// TIA Portal V20 export
FUNCTION_BLOCK "Sequence_2_SepaGripper"   // FB228, LAD
AUTHOR : ERsystem_FA2_DH. Kim
// stored: IsIECCheckEnabled true, MemoryReserve 100, Namespace Unit1.Em7, SetENOAutomatically false
   VAR_INPUT
      unitStatus { ExternalAccessible := 'False'; ExternalVisible := 'False'; ExternalWritable := 'False'} : "LAF_typeUnitStatus";   // Current unit status o be used in this EM
   END_VAR
   VAR
      statSelectedJobNumber { ExternalWritable := 'False'} : DInt;   // Evaluated Job Number
      instSequenceLADStatus { ExternalWritable := 'False'} : "LAF_StatusLadSequence";
      instSequenceLADControl { ExternalWritable := 'False'} : "LAF_ControlLadSequence";
      statTonTime { ExternalAccessible := 'False'; ExternalVisible := 'False'; ExternalWritable := 'False'} : Array[0..999] of TON_TIME;
   END_VAR
   VAR CONSTANT
      STEP_IDLE : DInt := 1;
      STEP_IMMEDIATE_STOP : DInt := 9001;   // Step executed when an immediate stop command is triggered for the sequence (i.e. when unit is in state aborting)
      JOB_1_STEP_01 : DInt := 101;
      JOB_1_STEP_10 : DInt := 110;
      JOB_1_STEP_20 : DInt := 120;
      JOB_1_STEP_30 : DInt := 130;
      JOB_1_STEP_40 : DInt := 140;
      JOB_1_STEP_41 : DInt := 141;
      JOB_1_STEP_50 : DInt := 150;
      JOB_1_STEP_80 : DInt := 180;
      JOB_1_STEP_90 : DInt := 190;
      JOB_2_STEP_01 : DInt := 201;
      JOB_2_STEP_10 : DInt := 210;
      JOB_2_STEP_20 : DInt := 220;
      JOB_2_STEP_30 : DInt := 230;
      JOB_2_STEP_31 : DInt := 231;
      JOB_2_STEP_40 : DInt := 240;
      JOB_2_STEP_50 : DInt := 250;
      JOB_2_STEP_51 : DInt := 251;
      JOB_2_STEP_80 : DInt := 280;
      JOB_2_STEP_90 : DInt := 290;
      JOB_3_STEP_01 : DInt := 301;
      JOB_3_STEP_10 : DInt := 310;
      JOB_3_STEP_11 : DInt := 311;
      JOB_3_STEP_20 : DInt := 320;
      JOB_3_STEP_30 : DInt := 330;
      JOB_3_STEP_31 : DInt := 331;
      JOB_3_STEP_90 : DInt := 390;
      JOB_4_STEP_01 : DInt := 401;
      JOB_4_STEP_10 : DInt := 410;
      JOB_4_STEP_20 : DInt := 420;
      JOB_4_STEP_21 : DInt := 421;
      JOB_4_STEP_30 : DInt := 430;
      JOB_4_STEP_90 : DInt := 490;
      JOB_5_STEP_01 : DInt := 501;
      JOB_5_STEP_10 : DInt := 510;
      JOB_5_STEP_20 : DInt := 520;
      JOB_5_STEP_30 : DInt := 530;
      JOB_5_STEP_31 : DInt := 531;
      JOB_5_STEP_40 : DInt := 540;
      JOB_5_STEP_50 : DInt := 550;
      JOB_5_STEP_80 : DInt := 580;
      JOB_5_STEP_81 : DInt := 581;
      JOB_5_STEP_90 : DInt := 590;
      JOB_6_STEP_01 : DInt := 601;
      JOB_6_STEP_10 : DInt := 610;
      JOB_6_STEP_11 : DInt := 611;
      JOB_6_STEP_20 : DInt := 620;
      JOB_6_STEP_90 : DInt := 690;
      JOB_7_STEP_01 : DInt := 701;
      JOB_7_STEP_10 : DInt := 710;
      JOB_7_STEP_20 : DInt := 720;
      JOB_7_STEP_30 : DInt := 730;
      JOB_7_STEP_40 : DInt := 740;
      JOB_7_STEP_50 : DInt := 750;
      JOB_7_STEP_90 : DInt := 790;
      JOB_8_STEP_01 : DInt := 801;
      JOB_8_STEP_10 : DInt := 810;
      JOB_8_STEP_11 : DInt := 811;
      JOB_8_STEP_20 : DInt := 820;
      JOB_8_STEP_21 : DInt := 821;
      JOB_8_STEP_30 : DInt := 830;
      JOB_8_STEP_31 : DInt := 831;
      JOB_8_STEP_90 : DInt := 890;
      JOB_9_STEP_01 : DInt := 901;
      JOB_9_STEP_10 : DInt := 910;
      JOB_9_STEP_20 : DInt := 920;
      JOB_9_STEP_30 : DInt := 930;
      JOB_9_STEP_40 : DInt := 940;
      JOB_9_STEP_50 : DInt := 950;
      JOB_9_STEP_90 : DInt := 990;
      JOB_11_STEP_01 : DInt := 1101;
      JOB_11_STEP_10 : DInt := 1110;
      JOB_11_STEP_20 : DInt := 1120;
      JOB_11_STEP_30 : DInt := 1130;
      JOB_11_STEP_40 : DInt := 1140;
      JOB_11_STEP_90 : DInt := 1190;
      JOB_12_STEP_01 : DInt := 1201;
      JOB_12_STEP_10 : DInt := 1210;
      JOB_12_STEP_11 : DInt := 1211;
      JOB_12_STEP_15 : DInt := 1215;
      JOB_12_STEP_16 : DInt := 1216;
      JOB_12_STEP_20 : DInt := 1220;
      JOB_12_STEP_30 : DInt := 1230;
      JOB_12_STEP_40 : DInt := 1240;
      JOB_12_STEP_90 : DInt := 1290;
      JOB_13_STEP_01 : DInt := 1301;
      JOB_13_STEP_10 : DInt := 1310;
      JOB_13_STEP_11 : DInt := 1311;
      JOB_13_STEP_90 : DInt := 1390;
      JOB_14_STEP_01 : DInt := 1401;
      JOB_14_STEP_10 : DInt := 1410;
      JOB_14_STEP_20 : DInt := 1420;
      JOB_14_STEP_90 : DInt := 1490;
      JOB_15_STEP_01 : DInt := 1501;
      JOB_15_STEP_10 : DInt := 1510;
      JOB_15_STEP_11 : DInt := 1511;
      JOB_15_STEP_20 : DInt := 1520;
      JOB_15_STEP_25 : DInt := 1525;
      JOB_15_STEP_30 : DInt := 1530;
      JOB_15_STEP_40 : DInt := 1540;
      JOB_15_STEP_50 : DInt := 1550;
      JOB_15_STEP_60 : DInt := 1560;
      JOB_15_STEP_70 : DInt := 1570;
      JOB_15_STEP_90 : DInt := 1590;
      JOB_16_STEP_01 : DInt := 1601;
      JOB_16_STEP_10 : DInt := 1610;
      JOB_16_STEP_20 : DInt := 1620;
      JOB_16_STEP_30 : DInt := 1630;
      JOB_16_STEP_40 : DInt := 1640;
      JOB_16_STEP_50 : DInt := 1650;
      JOB_16_STEP_90 : DInt := 1690;
      JOB_17_STEP_01 : DInt := 1701;
      JOB_17_STEP_10 : DInt := 1710;
      JOB_17_STEP_11 : DInt := 1711;
      JOB_17_STEP_20 : DInt := 1720;
      JOB_17_STEP_21 : DInt := 1721;
      JOB_17_STEP_30 : DInt := 1730;
      JOB_17_STEP_31 : DInt := 1731;
      JOB_17_STEP_90 : DInt := 1790;
      JOB_18_STEP_01 : DInt := 1801;
      JOB_18_STEP_10 : DInt := 1810;
      JOB_18_STEP_20 : DInt := 1820;
      JOB_18_STEP_30 : DInt := 1830;
      JOB_18_STEP_40 : DInt := 1840;
      JOB_18_STEP_50 : DInt := 1850;
      JOB_18_STEP_90 : DInt := 1890;
      FALSE : Bool := FALSE;
      TRUE : Bool := TRUE;
   END_VAR
   VAR_TEMP   // added for the SCL form of the ladder/FBD networks
      _w1 : Bool;
      _w2 : Bool;
   END_VAR
BEGIN

REGION Network 1: BLOCK INFO HEADER
   // (company) / (C) Copyright (year)
   // ---------------------------------------------------------------------------------
   // Title:                             (Title of this block)
   // Comment/Function: (that is implemented in the block)
   // Library/Family:           (that the source is dedicated to)
   // Author:                        (department / person in charge / contact)
   // Target System:          (test system with FW version)
   // Engineering:              TIA Portal (SW version)
   // Restrictions:               (OB types, etc.)
   // Requirements:           (hardware, technological package, etc.)
   // ---------------------------------------------------------------------------------
   // Change log table:
   // Version          | Date             | Signature      | Expert in charge  | Changes applied ------------------------|----------------------|-------------------------|--------------------------------|-----------------------
   // 001.000.000 | yyyy-mm-dd | 0x00000000 | (name of expert) | First released version
END_REGION

REGION Network 2: DESCRIPTION
   // This is a template block provided by the Automation Framework. It can be used to create an own project.
   // The Block Info Header is prepared to put in your own data.
   // Description of the block could be added here and the docu created by Code2Docu.
END_REGION

REGION Network 3: ********************* CONTROL *************************
END_REGION

REGION Network 4: Sequence Control
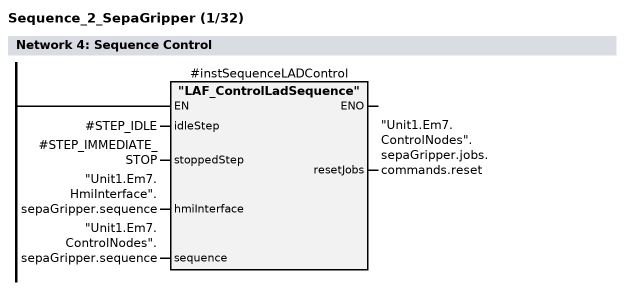
   RUNG wire#powerrail
      #instSequenceLADControl(idleStep := #STEP_IDLE, stoppedStep := #STEP_IMMEDIATE_STOP, hmiInterface := "Unit1.Em7.HmiInterface".sepaGripper.sequence, sequence := "Unit1.Em7.ControlNodes".sepaGripper.sequence, resetJobs => "Unit1.Em7.ControlNodes".sepaGripper.jobs.commands.reset)
   END_RUNG
   // the same network as SCL:
   #instSequenceLADControl(idleStep := #STEP_IDLE,   // "LAF_ControlLadSequence"
                           stoppedStep := #STEP_IMMEDIATE_STOP,
                           hmiInterface := "Unit1.Em7.HmiInterface".sepaGripper.sequence,
                           sequence := "Unit1.Em7.ControlNodes".sepaGripper.sequence,
                           resetJobs => "Unit1.Em7.ControlNodes".sepaGripper.jobs.commands.reset);
END_REGION

REGION Network 5: *************** JOB SELECT **************************
END_REGION

REGION Network 6: STEP IDLE
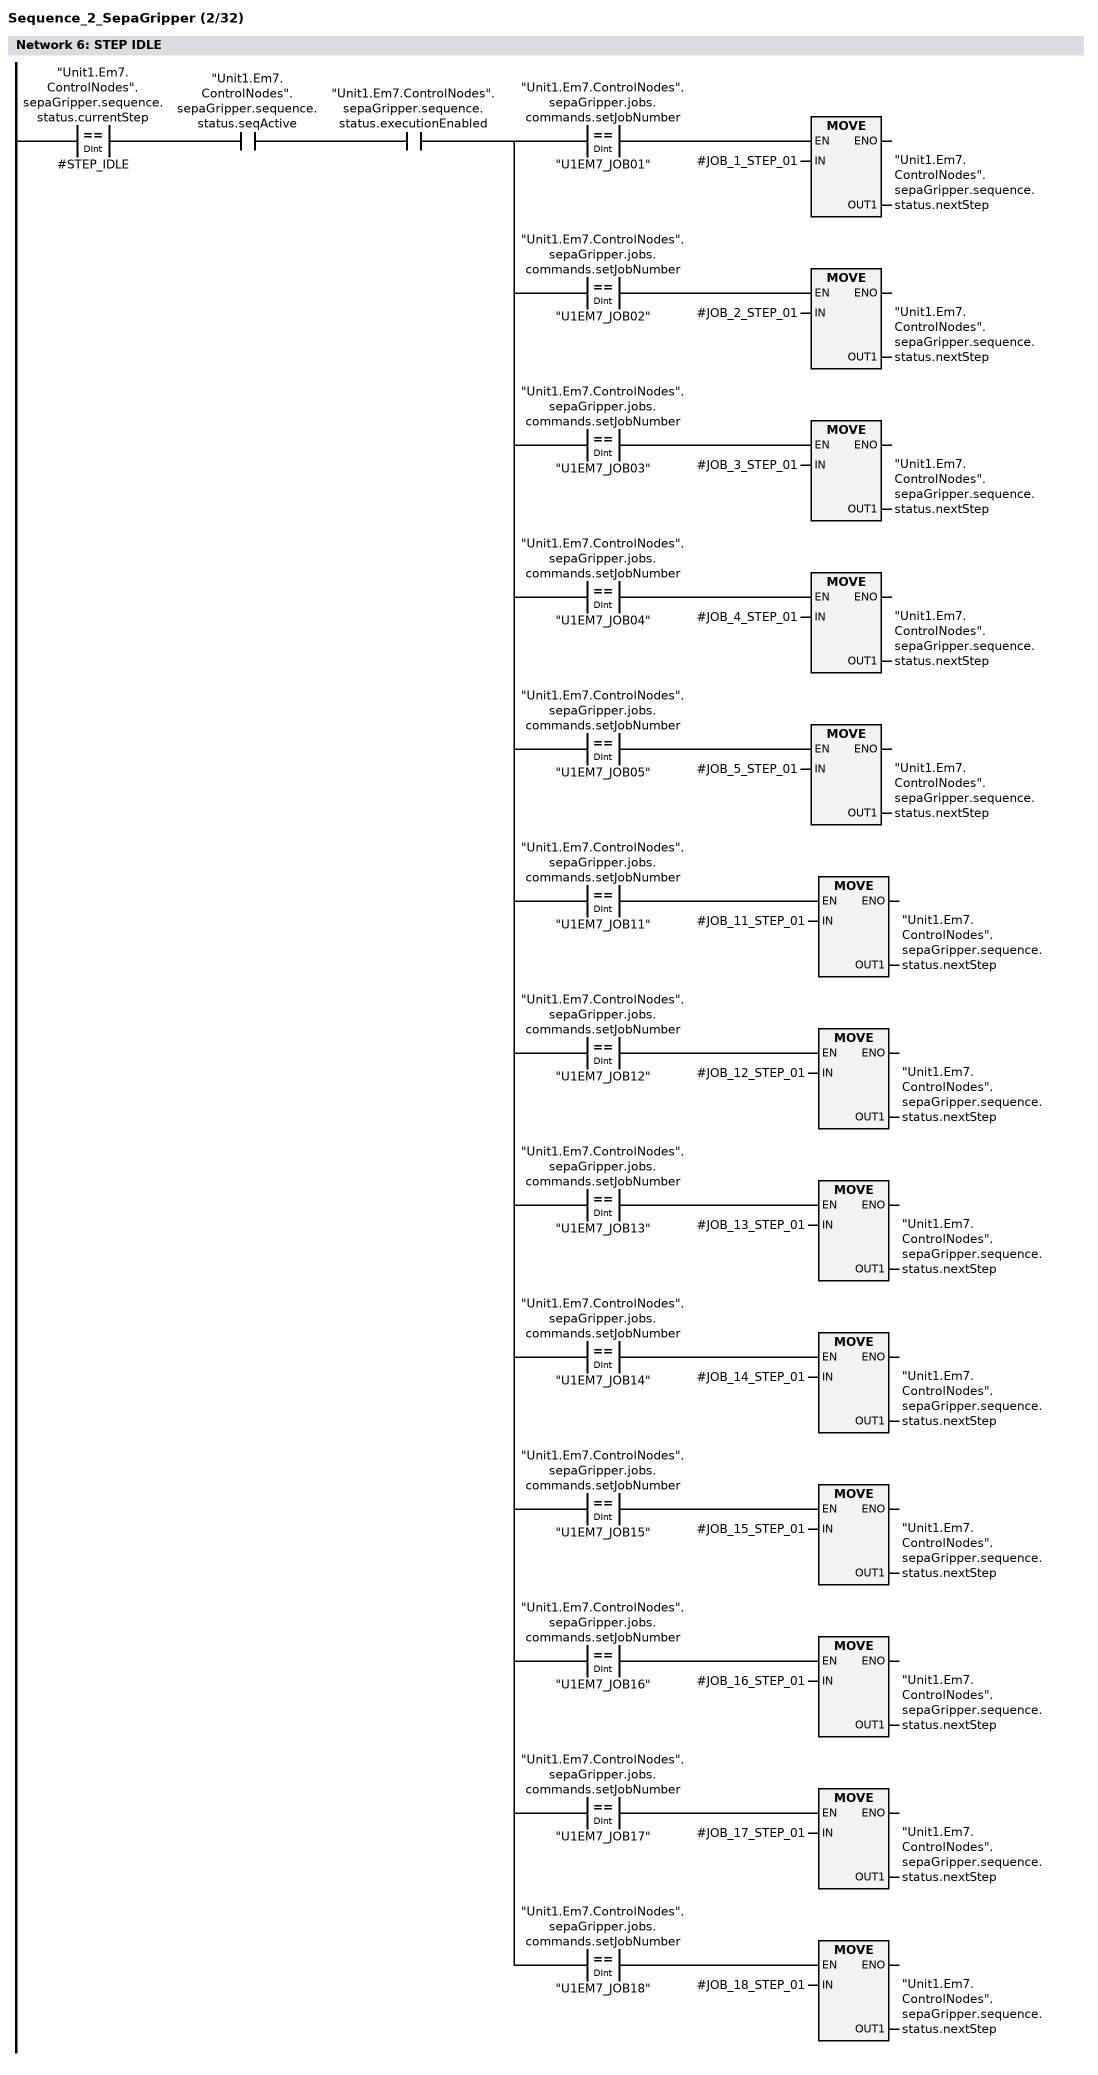
   RUNG wire#powerrail
      { S7_Templates := "SrcType := DInt" } EQ_Contact(in1 := "Unit1.Em7.ControlNodes".sepaGripper.sequence.status.currentStep, in2 := #STEP_IDLE)
      Contact( "Unit1.Em7.ControlNodes".sepaGripper.sequence.status.seqActive )
      Contact( "Unit1.Em7.ControlNodes".sepaGripper.sequence.status.executionEnabled )
      wire#w1
      { S7_Templates := "SrcType := DInt" } EQ_Contact(in1 := "Unit1.Em7.ControlNodes".sepaGripper.jobs.commands.setJobNumber, in2 := "U1EM7_JOB01")
      Move(in := #JOB_1_STEP_01, out1 => "Unit1.Em7.ControlNodes".sepaGripper.sequence.status.nextStep)
   END_RUNG
   RUNG wire#w1
      { S7_Templates := "SrcType := DInt" } EQ_Contact(in1 := "Unit1.Em7.ControlNodes".sepaGripper.jobs.commands.setJobNumber, in2 := "U1EM7_JOB02")
      Move(in := #JOB_2_STEP_01, out1 => "Unit1.Em7.ControlNodes".sepaGripper.sequence.status.nextStep)
   END_RUNG
   RUNG wire#w1
      { S7_Templates := "SrcType := DInt" } EQ_Contact(in1 := "Unit1.Em7.ControlNodes".sepaGripper.jobs.commands.setJobNumber, in2 := "U1EM7_JOB03")
      Move(in := #JOB_3_STEP_01, out1 => "Unit1.Em7.ControlNodes".sepaGripper.sequence.status.nextStep)
   END_RUNG
   RUNG wire#w1
      { S7_Templates := "SrcType := DInt" } EQ_Contact(in1 := "Unit1.Em7.ControlNodes".sepaGripper.jobs.commands.setJobNumber, in2 := "U1EM7_JOB04")
      Move(in := #JOB_4_STEP_01, out1 => "Unit1.Em7.ControlNodes".sepaGripper.sequence.status.nextStep)
   END_RUNG
   RUNG wire#w1
      { S7_Templates := "SrcType := DInt" } EQ_Contact(in1 := "Unit1.Em7.ControlNodes".sepaGripper.jobs.commands.setJobNumber, in2 := "U1EM7_JOB05")
      Move(in := #JOB_5_STEP_01, out1 => "Unit1.Em7.ControlNodes".sepaGripper.sequence.status.nextStep)
   END_RUNG
   RUNG wire#w1
      { S7_Templates := "SrcType := DInt" } EQ_Contact(in1 := "Unit1.Em7.ControlNodes".sepaGripper.jobs.commands.setJobNumber, in2 := "U1EM7_JOB11")
      Move(in := #JOB_11_STEP_01, out1 => "Unit1.Em7.ControlNodes".sepaGripper.sequence.status.nextStep)
   END_RUNG
   RUNG wire#w1
      { S7_Templates := "SrcType := DInt" } EQ_Contact(in1 := "Unit1.Em7.ControlNodes".sepaGripper.jobs.commands.setJobNumber, in2 := "U1EM7_JOB12")
      Move(in := #JOB_12_STEP_01, out1 => "Unit1.Em7.ControlNodes".sepaGripper.sequence.status.nextStep)
   END_RUNG
   RUNG wire#w1
      { S7_Templates := "SrcType := DInt" } EQ_Contact(in1 := "Unit1.Em7.ControlNodes".sepaGripper.jobs.commands.setJobNumber, in2 := "U1EM7_JOB13")
      Move(in := #JOB_13_STEP_01, out1 => "Unit1.Em7.ControlNodes".sepaGripper.sequence.status.nextStep)
   END_RUNG
   RUNG wire#w1
      { S7_Templates := "SrcType := DInt" } EQ_Contact(in1 := "Unit1.Em7.ControlNodes".sepaGripper.jobs.commands.setJobNumber, in2 := "U1EM7_JOB14")
      Move(in := #JOB_14_STEP_01, out1 => "Unit1.Em7.ControlNodes".sepaGripper.sequence.status.nextStep)
   END_RUNG
   RUNG wire#w1
      { S7_Templates := "SrcType := DInt" } EQ_Contact(in1 := "Unit1.Em7.ControlNodes".sepaGripper.jobs.commands.setJobNumber, in2 := "U1EM7_JOB15")
      Move(in := #JOB_15_STEP_01, out1 => "Unit1.Em7.ControlNodes".sepaGripper.sequence.status.nextStep)
   END_RUNG
   RUNG wire#w1
      { S7_Templates := "SrcType := DInt" } EQ_Contact(in1 := "Unit1.Em7.ControlNodes".sepaGripper.jobs.commands.setJobNumber, in2 := "U1EM7_JOB16")
      Move(in := #JOB_16_STEP_01, out1 => "Unit1.Em7.ControlNodes".sepaGripper.sequence.status.nextStep)
   END_RUNG
   RUNG wire#w1
      { S7_Templates := "SrcType := DInt" } EQ_Contact(in1 := "Unit1.Em7.ControlNodes".sepaGripper.jobs.commands.setJobNumber, in2 := "U1EM7_JOB17")
      Move(in := #JOB_17_STEP_01, out1 => "Unit1.Em7.ControlNodes".sepaGripper.sequence.status.nextStep)
   END_RUNG
   RUNG wire#w1
      { S7_Templates := "SrcType := DInt" } EQ_Contact(in1 := "Unit1.Em7.ControlNodes".sepaGripper.jobs.commands.setJobNumber, in2 := "U1EM7_JOB18")
      Move(in := #JOB_18_STEP_01, out1 => "Unit1.Em7.ControlNodes".sepaGripper.sequence.status.nextStep)
   END_RUNG
   // the same network as SCL:
   #_w1 := ("Unit1.Em7.ControlNodes".sepaGripper.sequence.status.currentStep = #STEP_IDLE) AND "Unit1.Em7.ControlNodes".sepaGripper.sequence.status.seqActive AND "Unit1.Em7.ControlNodes".sepaGripper.sequence.status.executionEnabled;
   IF #_w1 AND ("Unit1.Em7.ControlNodes".sepaGripper.jobs.commands.setJobNumber = "U1EM7_JOB01") THEN
       "Unit1.Em7.ControlNodes".sepaGripper.sequence.status.nextStep := #JOB_1_STEP_01;
   END_IF;
   IF #_w1 AND ("Unit1.Em7.ControlNodes".sepaGripper.jobs.commands.setJobNumber = "U1EM7_JOB02") THEN
       "Unit1.Em7.ControlNodes".sepaGripper.sequence.status.nextStep := #JOB_2_STEP_01;
   END_IF;
   IF #_w1 AND ("Unit1.Em7.ControlNodes".sepaGripper.jobs.commands.setJobNumber = "U1EM7_JOB03") THEN
       "Unit1.Em7.ControlNodes".sepaGripper.sequence.status.nextStep := #JOB_3_STEP_01;
   END_IF;
   IF #_w1 AND ("Unit1.Em7.ControlNodes".sepaGripper.jobs.commands.setJobNumber = "U1EM7_JOB04") THEN
       "Unit1.Em7.ControlNodes".sepaGripper.sequence.status.nextStep := #JOB_4_STEP_01;
   END_IF;
   IF #_w1 AND ("Unit1.Em7.ControlNodes".sepaGripper.jobs.commands.setJobNumber = "U1EM7_JOB05") THEN
       "Unit1.Em7.ControlNodes".sepaGripper.sequence.status.nextStep := #JOB_5_STEP_01;
   END_IF;
   IF #_w1 AND ("Unit1.Em7.ControlNodes".sepaGripper.jobs.commands.setJobNumber = "U1EM7_JOB11") THEN
       "Unit1.Em7.ControlNodes".sepaGripper.sequence.status.nextStep := #JOB_11_STEP_01;
   END_IF;
   IF #_w1 AND ("Unit1.Em7.ControlNodes".sepaGripper.jobs.commands.setJobNumber = "U1EM7_JOB12") THEN
       "Unit1.Em7.ControlNodes".sepaGripper.sequence.status.nextStep := #JOB_12_STEP_01;
   END_IF;
   IF #_w1 AND ("Unit1.Em7.ControlNodes".sepaGripper.jobs.commands.setJobNumber = "U1EM7_JOB13") THEN
       "Unit1.Em7.ControlNodes".sepaGripper.sequence.status.nextStep := #JOB_13_STEP_01;
   END_IF;
   IF #_w1 AND ("Unit1.Em7.ControlNodes".sepaGripper.jobs.commands.setJobNumber = "U1EM7_JOB14") THEN
       "Unit1.Em7.ControlNodes".sepaGripper.sequence.status.nextStep := #JOB_14_STEP_01;
   END_IF;
   IF #_w1 AND ("Unit1.Em7.ControlNodes".sepaGripper.jobs.commands.setJobNumber = "U1EM7_JOB15") THEN
       "Unit1.Em7.ControlNodes".sepaGripper.sequence.status.nextStep := #JOB_15_STEP_01;
   END_IF;
   IF #_w1 AND ("Unit1.Em7.ControlNodes".sepaGripper.jobs.commands.setJobNumber = "U1EM7_JOB16") THEN
       "Unit1.Em7.ControlNodes".sepaGripper.sequence.status.nextStep := #JOB_16_STEP_01;
   END_IF;
   IF #_w1 AND ("Unit1.Em7.ControlNodes".sepaGripper.jobs.commands.setJobNumber = "U1EM7_JOB17") THEN
       "Unit1.Em7.ControlNodes".sepaGripper.sequence.status.nextStep := #JOB_17_STEP_01;
   END_IF;
   IF #_w1 AND ("Unit1.Em7.ControlNodes".sepaGripper.jobs.commands.setJobNumber = "U1EM7_JOB18") THEN
       "Unit1.Em7.ControlNodes".sepaGripper.sequence.status.nextStep := #JOB_18_STEP_01;
   END_IF;
END_REGION

REGION Network 7: *************** JOB[1] EM HOMING ************************
END_REGION

REGION Network 8: Step[101] : JOB [Homing] Condition
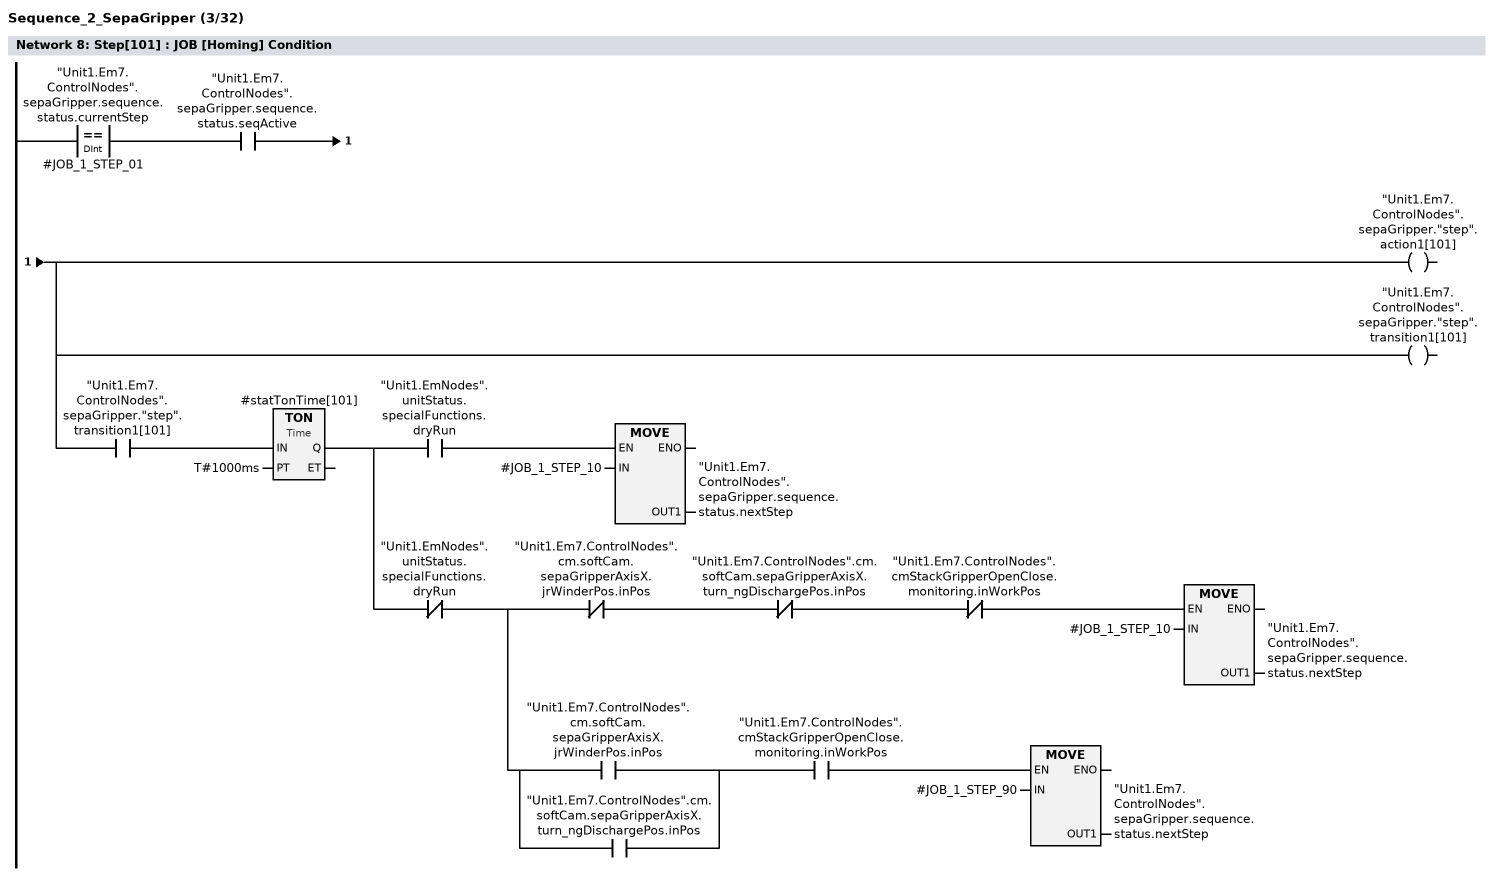
   RUNG wire#powerrail
      { S7_Templates := "SrcType := DInt" } EQ_Contact(in1 := "Unit1.Em7.ControlNodes".sepaGripper.sequence.status.currentStep, in2 := #JOB_1_STEP_01)
      Contact( "Unit1.Em7.ControlNodes".sepaGripper.sequence.status.seqActive )
      wire#w1
      Coil( "Unit1.Em7.ControlNodes".sepaGripper."step".action1[101] )
   END_RUNG
   RUNG wire#w1
      Coil( "Unit1.Em7.ControlNodes".sepaGripper."step".transition1[101] )
   END_RUNG
   RUNG wire#w1
      Contact( "Unit1.Em7.ControlNodes".sepaGripper."step".transition1[101] )
      { S7_Templates := "time_type := Time" } #statTonTime[101].TON(pt := T#1000ms, et =>)
      wire#w2
      Contact( "Unit1.EmNodes".unitStatus.specialFunctions.dryRun )
      Move(in := #JOB_1_STEP_10, out1 => "Unit1.Em7.ControlNodes".sepaGripper.sequence.status.nextStep)
   END_RUNG
   RUNG wire#w2
      I_Contact( "Unit1.EmNodes".unitStatus.specialFunctions.dryRun )
      wire#w3
      I_Contact( "Unit1.Em7.ControlNodes".cm.softCam.sepaGripperAxisX.jrWinderPos.inPos )
      I_Contact( "Unit1.Em7.ControlNodes".cm.softCam.sepaGripperAxisX.turn_ngDischargePos.inPos )
      I_Contact( "Unit1.Em7.ControlNodes".cmStackGripperOpenClose.monitoring.inWorkPos )
      Move(in := #JOB_1_STEP_10, out1 => "Unit1.Em7.ControlNodes".sepaGripper.sequence.status.nextStep)
   END_RUNG
   RUNG wire#w3
      Contact( "Unit1.Em7.ControlNodes".cm.softCam.sepaGripperAxisX.jrWinderPos.inPos )
      wire#w4
      Contact( "Unit1.Em7.ControlNodes".cmStackGripperOpenClose.monitoring.inWorkPos )
      Move(in := #JOB_1_STEP_90, out1 => "Unit1.Em7.ControlNodes".sepaGripper.sequence.status.nextStep)
   END_RUNG
   RUNG wire#w3
      Contact( "Unit1.Em7.ControlNodes".cm.softCam.sepaGripperAxisX.turn_ngDischargePos.inPos )
   END_RUNG wire#w4
   // the same network as SCL:
   "Unit1.Em7.ControlNodes".sepaGripper."step".action1[101] := ("Unit1.Em7.ControlNodes".sepaGripper.sequence.status.currentStep = #JOB_1_STEP_01) AND "Unit1.Em7.ControlNodes".sepaGripper.sequence.status.seqActive;
   "Unit1.Em7.ControlNodes".sepaGripper."step".transition1[101] := ("Unit1.Em7.ControlNodes".sepaGripper.sequence.status.currentStep = #JOB_1_STEP_01) AND "Unit1.Em7.ControlNodes".sepaGripper.sequence.status.seqActive;
   #statTonTime[101].TON(IN := ("Unit1.Em7.ControlNodes".sepaGripper.sequence.status.currentStep = #JOB_1_STEP_01) AND "Unit1.Em7.ControlNodes".sepaGripper.sequence.status.seqActive AND "Unit1.Em7.ControlNodes".sepaGripper."step".transition1[101],
                         PT := T#1000ms);
   IF #statTonTime[101].Q AND "Unit1.EmNodes".unitStatus.specialFunctions.dryRun THEN
       "Unit1.Em7.ControlNodes".sepaGripper.sequence.status.nextStep := #JOB_1_STEP_10;
   END_IF;
   #_w1 := #statTonTime[101].Q AND NOT "Unit1.EmNodes".unitStatus.specialFunctions.dryRun;
   IF #_w1 AND NOT "Unit1.Em7.ControlNodes".cm.softCam.sepaGripperAxisX.jrWinderPos.inPos AND NOT "Unit1.Em7.ControlNodes".cm.softCam.sepaGripperAxisX.turn_ngDischargePos.inPos AND NOT "Unit1.Em7.ControlNodes".cmStackGripperOpenClose.monitoring.inWorkPos THEN
       "Unit1.Em7.ControlNodes".sepaGripper.sequence.status.nextStep := #JOB_1_STEP_10;
   END_IF;
   IF #_w1 AND ("Unit1.Em7.ControlNodes".cm.softCam.sepaGripperAxisX.jrWinderPos.inPos OR "Unit1.Em7.ControlNodes".cm.softCam.sepaGripperAxisX.turn_ngDischargePos.inPos) AND "Unit1.Em7.ControlNodes".cmStackGripperOpenClose.monitoring.inWorkPos THEN
       "Unit1.Em7.ControlNodes".sepaGripper.sequence.status.nextStep := #JOB_1_STEP_90;
   END_IF;
END_REGION

REGION Network 9: Step[110] : Gripper Open
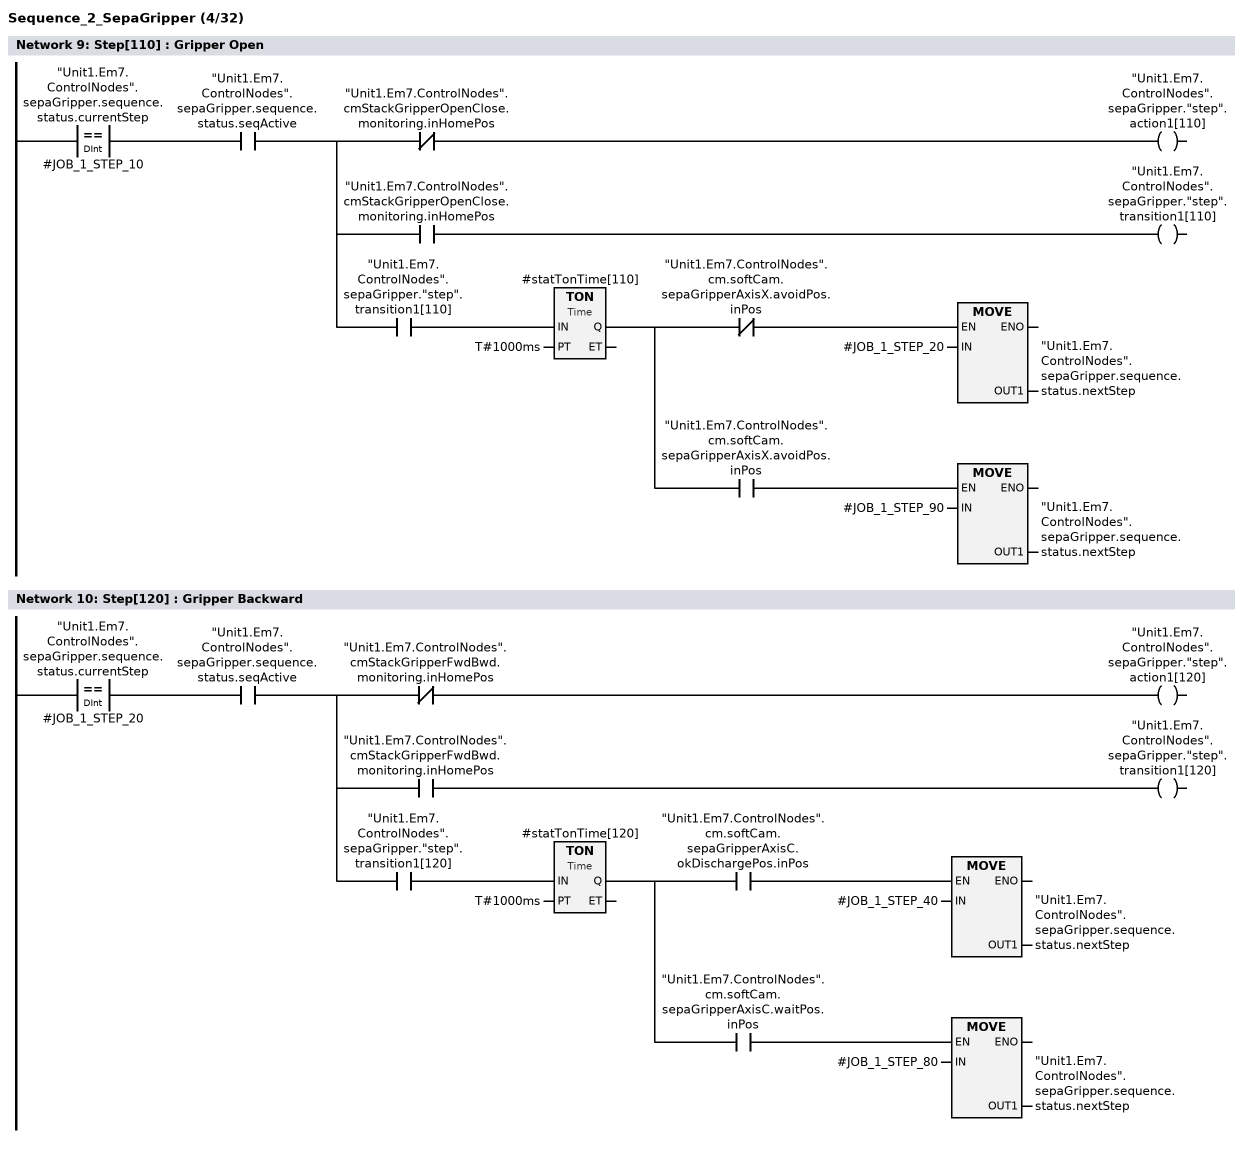
   RUNG wire#powerrail
      { S7_Templates := "SrcType := DInt" } EQ_Contact(in1 := "Unit1.Em7.ControlNodes".sepaGripper.sequence.status.currentStep, in2 := #JOB_1_STEP_10)
      Contact( "Unit1.Em7.ControlNodes".sepaGripper.sequence.status.seqActive )
      wire#w1
      I_Contact( "Unit1.Em7.ControlNodes".cmStackGripperOpenClose.monitoring.inHomePos )
      Coil( "Unit1.Em7.ControlNodes".sepaGripper."step".action1[110] )
   END_RUNG
   RUNG wire#w1
      Contact( "Unit1.Em7.ControlNodes".cmStackGripperOpenClose.monitoring.inHomePos )
      Coil( "Unit1.Em7.ControlNodes".sepaGripper."step".transition1[110] )
   END_RUNG
   RUNG wire#w1
      Contact( "Unit1.Em7.ControlNodes".sepaGripper."step".transition1[110] )
      { S7_Templates := "time_type := Time" } #statTonTime[110].TON(pt := T#1000ms, et =>)
      wire#w2
      I_Contact( "Unit1.Em7.ControlNodes".cm.softCam.sepaGripperAxisX.avoidPos.inPos )
      Move(in := #JOB_1_STEP_20, out1 => "Unit1.Em7.ControlNodes".sepaGripper.sequence.status.nextStep)
   END_RUNG
   RUNG wire#w2
      Contact( "Unit1.Em7.ControlNodes".cm.softCam.sepaGripperAxisX.avoidPos.inPos )
      Move(in := #JOB_1_STEP_90, out1 => "Unit1.Em7.ControlNodes".sepaGripper.sequence.status.nextStep)
   END_RUNG
   // the same network as SCL:
   #_w1 := ("Unit1.Em7.ControlNodes".sepaGripper.sequence.status.currentStep = #JOB_1_STEP_10) AND "Unit1.Em7.ControlNodes".sepaGripper.sequence.status.seqActive;
   "Unit1.Em7.ControlNodes".sepaGripper."step".action1[110] := #_w1 AND NOT "Unit1.Em7.ControlNodes".cmStackGripperOpenClose.monitoring.inHomePos;
   "Unit1.Em7.ControlNodes".sepaGripper."step".transition1[110] := #_w1 AND "Unit1.Em7.ControlNodes".cmStackGripperOpenClose.monitoring.inHomePos;
   #statTonTime[110].TON(IN := #_w1 AND "Unit1.Em7.ControlNodes".sepaGripper."step".transition1[110],
                         PT := T#1000ms);
   IF #statTonTime[110].Q AND NOT "Unit1.Em7.ControlNodes".cm.softCam.sepaGripperAxisX.avoidPos.inPos THEN
       "Unit1.Em7.ControlNodes".sepaGripper.sequence.status.nextStep := #JOB_1_STEP_20;
   END_IF;
   IF #statTonTime[110].Q AND "Unit1.Em7.ControlNodes".cm.softCam.sepaGripperAxisX.avoidPos.inPos THEN
       "Unit1.Em7.ControlNodes".sepaGripper.sequence.status.nextStep := #JOB_1_STEP_90;
   END_IF;
END_REGION

REGION Network 10: Step[120] : Gripper Backward
   RUNG wire#powerrail
      { S7_Templates := "SrcType := DInt" } EQ_Contact(in1 := "Unit1.Em7.ControlNodes".sepaGripper.sequence.status.currentStep, in2 := #JOB_1_STEP_20)
      Contact( "Unit1.Em7.ControlNodes".sepaGripper.sequence.status.seqActive )
      wire#w1
      I_Contact( "Unit1.Em7.ControlNodes".cmStackGripperFwdBwd.monitoring.inHomePos )
      Coil( "Unit1.Em7.ControlNodes".sepaGripper."step".action1[120] )
   END_RUNG
   RUNG wire#w1
      Contact( "Unit1.Em7.ControlNodes".cmStackGripperFwdBwd.monitoring.inHomePos )
      Coil( "Unit1.Em7.ControlNodes".sepaGripper."step".transition1[120] )
   END_RUNG
   RUNG wire#w1
      Contact( "Unit1.Em7.ControlNodes".sepaGripper."step".transition1[120] )
      { S7_Templates := "time_type := Time" } #statTonTime[120].TON(pt := T#1000ms, et =>)
      wire#w2
      Contact( "Unit1.Em7.ControlNodes".cm.softCam.sepaGripperAxisC.okDischargePos.inPos )
      Move(in := #JOB_1_STEP_40, out1 => "Unit1.Em7.ControlNodes".sepaGripper.sequence.status.nextStep)
   END_RUNG
   RUNG wire#w2
      Contact( "Unit1.Em7.ControlNodes".cm.softCam.sepaGripperAxisC.waitPos.inPos )
      Move(in := #JOB_1_STEP_80, out1 => "Unit1.Em7.ControlNodes".sepaGripper.sequence.status.nextStep)
   END_RUNG
   // the same network as SCL:
   #_w1 := ("Unit1.Em7.ControlNodes".sepaGripper.sequence.status.currentStep = #JOB_1_STEP_20) AND "Unit1.Em7.ControlNodes".sepaGripper.sequence.status.seqActive;
   "Unit1.Em7.ControlNodes".sepaGripper."step".action1[120] := #_w1 AND NOT "Unit1.Em7.ControlNodes".cmStackGripperFwdBwd.monitoring.inHomePos;
   "Unit1.Em7.ControlNodes".sepaGripper."step".transition1[120] := #_w1 AND "Unit1.Em7.ControlNodes".cmStackGripperFwdBwd.monitoring.inHomePos;
   #statTonTime[120].TON(IN := #_w1 AND "Unit1.Em7.ControlNodes".sepaGripper."step".transition1[120],
                         PT := T#1000ms);
   IF #statTonTime[120].Q AND "Unit1.Em7.ControlNodes".cm.softCam.sepaGripperAxisC.okDischargePos.inPos THEN
       "Unit1.Em7.ControlNodes".sepaGripper.sequence.status.nextStep := #JOB_1_STEP_40;
   END_IF;
   IF #statTonTime[120].Q AND "Unit1.Em7.ControlNodes".cm.softCam.sepaGripperAxisC.waitPos.inPos THEN
       "Unit1.Em7.ControlNodes".sepaGripper.sequence.status.nextStep := #JOB_1_STEP_80;
   END_IF;
END_REGION

REGION Network 11: Step[140] : Gripper X-Axis Turn Pos
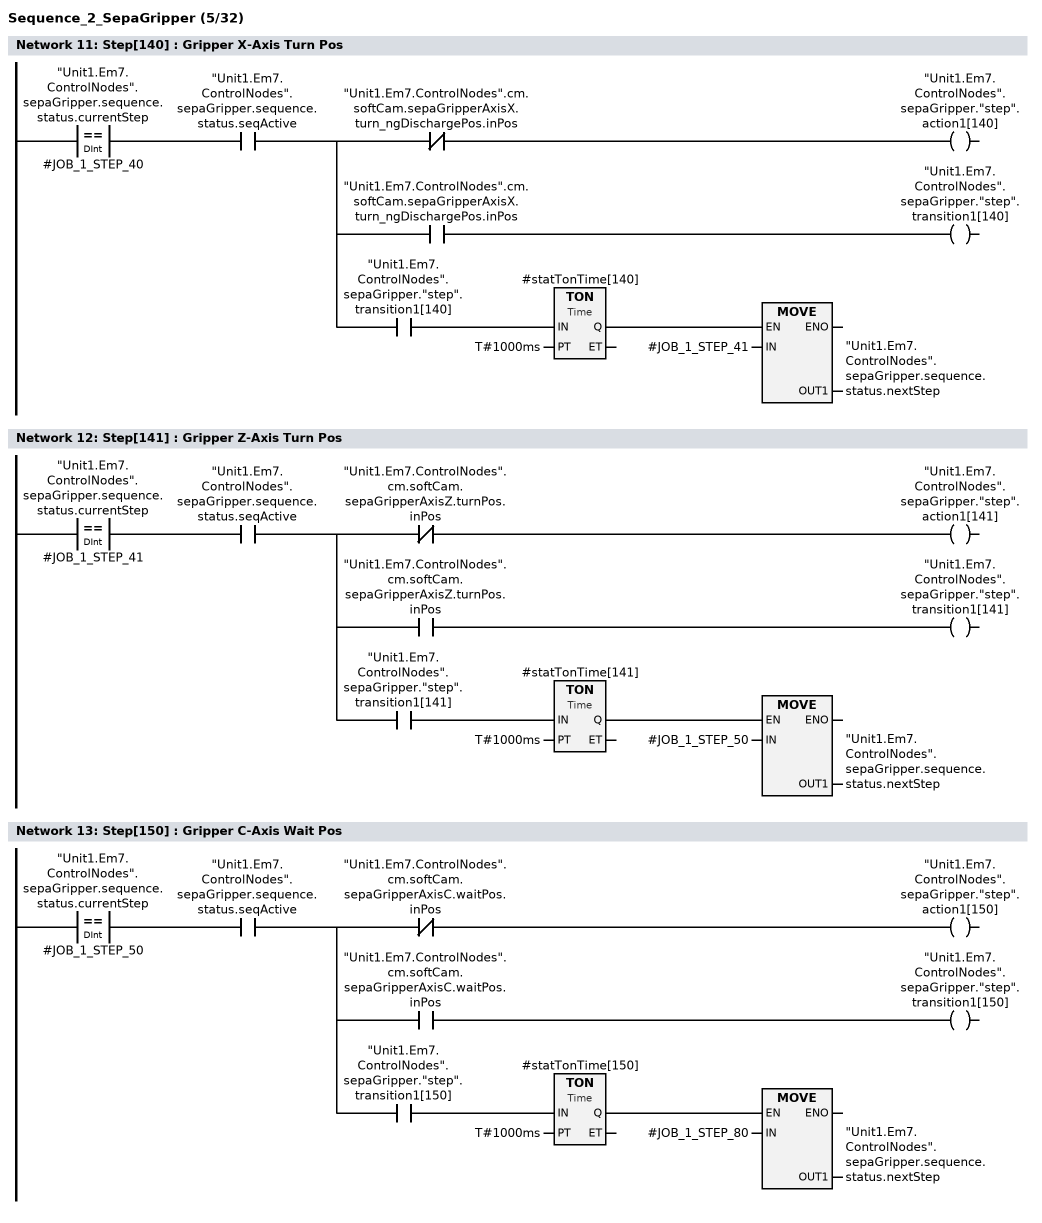
   RUNG wire#powerrail
      { S7_Templates := "SrcType := DInt" } EQ_Contact(in1 := "Unit1.Em7.ControlNodes".sepaGripper.sequence.status.currentStep, in2 := #JOB_1_STEP_40)
      Contact( "Unit1.Em7.ControlNodes".sepaGripper.sequence.status.seqActive )
      wire#w1
      I_Contact( "Unit1.Em7.ControlNodes".cm.softCam.sepaGripperAxisX.turn_ngDischargePos.inPos )
      Coil( "Unit1.Em7.ControlNodes".sepaGripper."step".action1[140] )
   END_RUNG
   RUNG wire#w1
      Contact( "Unit1.Em7.ControlNodes".cm.softCam.sepaGripperAxisX.turn_ngDischargePos.inPos )
      Coil( "Unit1.Em7.ControlNodes".sepaGripper."step".transition1[140] )
   END_RUNG
   RUNG wire#w1
      Contact( "Unit1.Em7.ControlNodes".sepaGripper."step".transition1[140] )
      { S7_Templates := "time_type := Time" } #statTonTime[140].TON(pt := T#1000ms, et =>)
      Move(in := #JOB_1_STEP_41, out1 => "Unit1.Em7.ControlNodes".sepaGripper.sequence.status.nextStep)
   END_RUNG
   // the same network as SCL:
   #_w1 := ("Unit1.Em7.ControlNodes".sepaGripper.sequence.status.currentStep = #JOB_1_STEP_40) AND "Unit1.Em7.ControlNodes".sepaGripper.sequence.status.seqActive;
   "Unit1.Em7.ControlNodes".sepaGripper."step".action1[140] := #_w1 AND NOT "Unit1.Em7.ControlNodes".cm.softCam.sepaGripperAxisX.turn_ngDischargePos.inPos;
   "Unit1.Em7.ControlNodes".sepaGripper."step".transition1[140] := #_w1 AND "Unit1.Em7.ControlNodes".cm.softCam.sepaGripperAxisX.turn_ngDischargePos.inPos;
   #statTonTime[140].TON(IN := #_w1 AND "Unit1.Em7.ControlNodes".sepaGripper."step".transition1[140],
                         PT := T#1000ms);
   IF #statTonTime[140].Q THEN
       "Unit1.Em7.ControlNodes".sepaGripper.sequence.status.nextStep := #JOB_1_STEP_41;
   END_IF;
END_REGION

REGION Network 12: Step[141] : Gripper Z-Axis Turn Pos
   RUNG wire#powerrail
      { S7_Templates := "SrcType := DInt" } EQ_Contact(in1 := "Unit1.Em7.ControlNodes".sepaGripper.sequence.status.currentStep, in2 := #JOB_1_STEP_41)
      Contact( "Unit1.Em7.ControlNodes".sepaGripper.sequence.status.seqActive )
      wire#w1
      I_Contact( "Unit1.Em7.ControlNodes".cm.softCam.sepaGripperAxisZ.turnPos.inPos )
      Coil( "Unit1.Em7.ControlNodes".sepaGripper."step".action1[141] )
   END_RUNG
   RUNG wire#w1
      Contact( "Unit1.Em7.ControlNodes".cm.softCam.sepaGripperAxisZ.turnPos.inPos )
      Coil( "Unit1.Em7.ControlNodes".sepaGripper."step".transition1[141] )
   END_RUNG
   RUNG wire#w1
      Contact( "Unit1.Em7.ControlNodes".sepaGripper."step".transition1[141] )
      { S7_Templates := "time_type := Time" } #statTonTime[141].TON(pt := T#1000ms, et =>)
      Move(in := #JOB_1_STEP_50, out1 => "Unit1.Em7.ControlNodes".sepaGripper.sequence.status.nextStep)
   END_RUNG
   // the same network as SCL:
   #_w1 := ("Unit1.Em7.ControlNodes".sepaGripper.sequence.status.currentStep = #JOB_1_STEP_41) AND "Unit1.Em7.ControlNodes".sepaGripper.sequence.status.seqActive;
   "Unit1.Em7.ControlNodes".sepaGripper."step".action1[141] := #_w1 AND NOT "Unit1.Em7.ControlNodes".cm.softCam.sepaGripperAxisZ.turnPos.inPos;
   "Unit1.Em7.ControlNodes".sepaGripper."step".transition1[141] := #_w1 AND "Unit1.Em7.ControlNodes".cm.softCam.sepaGripperAxisZ.turnPos.inPos;
   #statTonTime[141].TON(IN := #_w1 AND "Unit1.Em7.ControlNodes".sepaGripper."step".transition1[141],
                         PT := T#1000ms);
   IF #statTonTime[141].Q THEN
       "Unit1.Em7.ControlNodes".sepaGripper.sequence.status.nextStep := #JOB_1_STEP_50;
   END_IF;
END_REGION

REGION Network 13: Step[150] : Gripper C-Axis Wait Pos
   RUNG wire#powerrail
      { S7_Templates := "SrcType := DInt" } EQ_Contact(in1 := "Unit1.Em7.ControlNodes".sepaGripper.sequence.status.currentStep, in2 := #JOB_1_STEP_50)
      Contact( "Unit1.Em7.ControlNodes".sepaGripper.sequence.status.seqActive )
      wire#w1
      I_Contact( "Unit1.Em7.ControlNodes".cm.softCam.sepaGripperAxisC.waitPos.inPos )
      Coil( "Unit1.Em7.ControlNodes".sepaGripper."step".action1[150] )
   END_RUNG
   RUNG wire#w1
      Contact( "Unit1.Em7.ControlNodes".cm.softCam.sepaGripperAxisC.waitPos.inPos )
      Coil( "Unit1.Em7.ControlNodes".sepaGripper."step".transition1[150] )
   END_RUNG
   RUNG wire#w1
      Contact( "Unit1.Em7.ControlNodes".sepaGripper."step".transition1[150] )
      { S7_Templates := "time_type := Time" } #statTonTime[150].TON(pt := T#1000ms, et =>)
      Move(in := #JOB_1_STEP_80, out1 => "Unit1.Em7.ControlNodes".sepaGripper.sequence.status.nextStep)
   END_RUNG
   // the same network as SCL:
   #_w1 := ("Unit1.Em7.ControlNodes".sepaGripper.sequence.status.currentStep = #JOB_1_STEP_50) AND "Unit1.Em7.ControlNodes".sepaGripper.sequence.status.seqActive;
   "Unit1.Em7.ControlNodes".sepaGripper."step".action1[150] := #_w1 AND NOT "Unit1.Em7.ControlNodes".cm.softCam.sepaGripperAxisC.waitPos.inPos;
   "Unit1.Em7.ControlNodes".sepaGripper."step".transition1[150] := #_w1 AND "Unit1.Em7.ControlNodes".cm.softCam.sepaGripperAxisC.waitPos.inPos;
   #statTonTime[150].TON(IN := #_w1 AND "Unit1.Em7.ControlNodes".sepaGripper."step".transition1[150],
                         PT := T#1000ms);
   IF #statTonTime[150].Q THEN
       "Unit1.Em7.ControlNodes".sepaGripper.sequence.status.nextStep := #JOB_1_STEP_80;
   END_IF;
END_REGION

REGION Network 14: Step[180] : Gripper X,Z-Axis Wait Pos
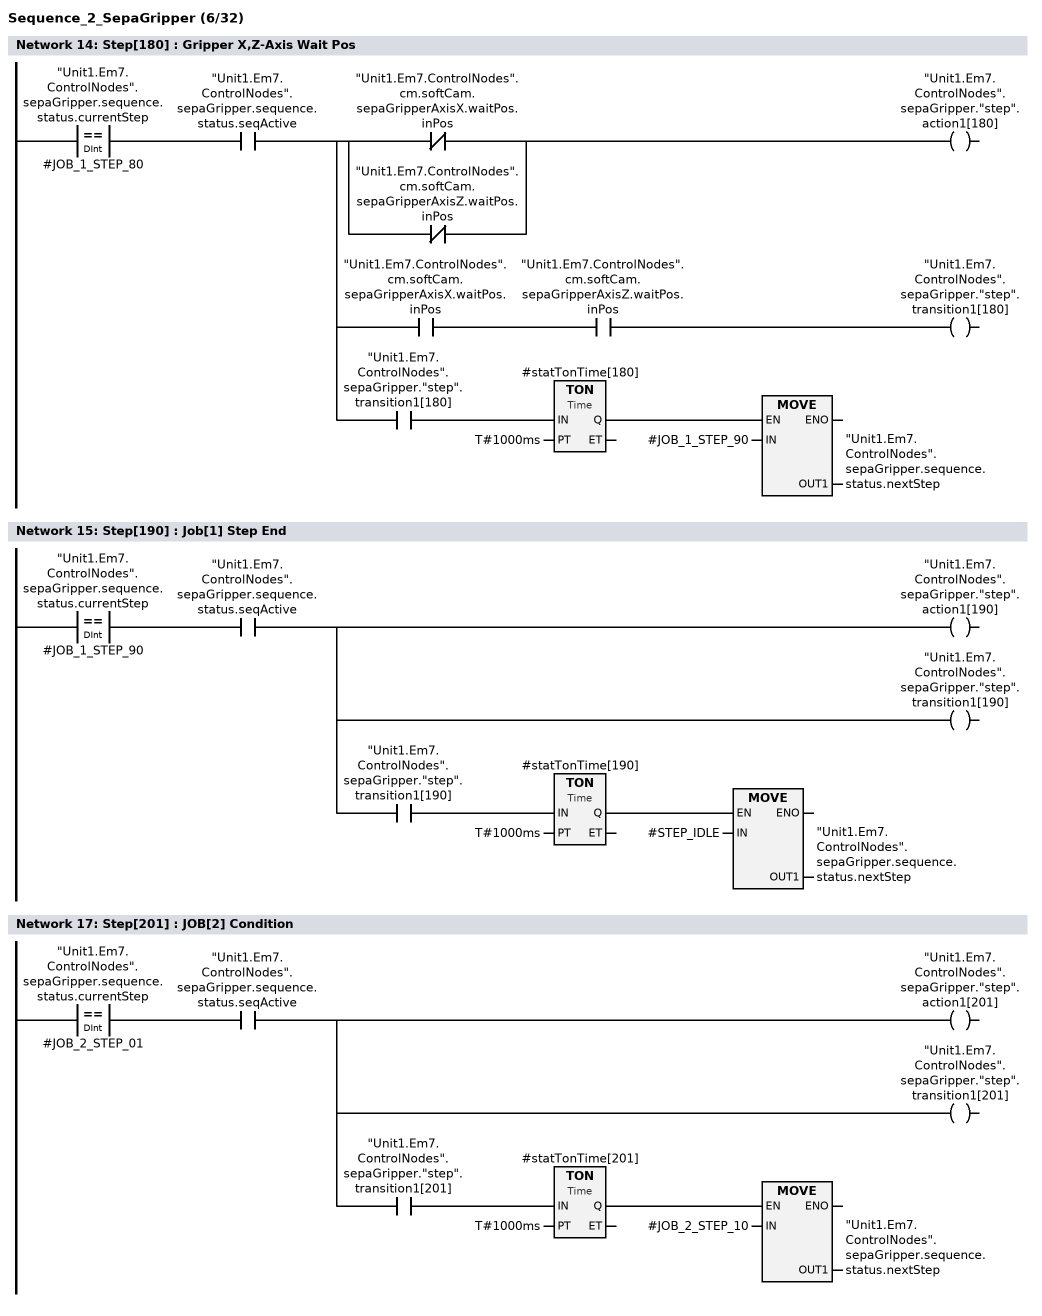
   RUNG wire#powerrail
      { S7_Templates := "SrcType := DInt" } EQ_Contact(in1 := "Unit1.Em7.ControlNodes".sepaGripper.sequence.status.currentStep, in2 := #JOB_1_STEP_80)
      Contact( "Unit1.Em7.ControlNodes".sepaGripper.sequence.status.seqActive )
      wire#w1
      I_Contact( "Unit1.Em7.ControlNodes".cm.softCam.sepaGripperAxisX.waitPos.inPos )
      wire#w2
      Coil( "Unit1.Em7.ControlNodes".sepaGripper."step".action1[180] )
   END_RUNG
   RUNG wire#w1
      I_Contact( "Unit1.Em7.ControlNodes".cm.softCam.sepaGripperAxisZ.waitPos.inPos )
   END_RUNG wire#w2
   RUNG wire#w1
      Contact( "Unit1.Em7.ControlNodes".cm.softCam.sepaGripperAxisX.waitPos.inPos )
      Contact( "Unit1.Em7.ControlNodes".cm.softCam.sepaGripperAxisZ.waitPos.inPos )
      Coil( "Unit1.Em7.ControlNodes".sepaGripper."step".transition1[180] )
   END_RUNG
   RUNG wire#w1
      Contact( "Unit1.Em7.ControlNodes".sepaGripper."step".transition1[180] )
      { S7_Templates := "time_type := Time" } #statTonTime[180].TON(pt := T#1000ms, et =>)
      Move(in := #JOB_1_STEP_90, out1 => "Unit1.Em7.ControlNodes".sepaGripper.sequence.status.nextStep)
   END_RUNG
   // the same network as SCL:
   #_w1 := ("Unit1.Em7.ControlNodes".sepaGripper.sequence.status.currentStep = #JOB_1_STEP_80) AND "Unit1.Em7.ControlNodes".sepaGripper.sequence.status.seqActive;
   "Unit1.Em7.ControlNodes".sepaGripper."step".action1[180] := #_w1 AND (NOT "Unit1.Em7.ControlNodes".cm.softCam.sepaGripperAxisX.waitPos.inPos OR NOT "Unit1.Em7.ControlNodes".cm.softCam.sepaGripperAxisZ.waitPos.inPos);
   "Unit1.Em7.ControlNodes".sepaGripper."step".transition1[180] := #_w1 AND "Unit1.Em7.ControlNodes".cm.softCam.sepaGripperAxisX.waitPos.inPos AND "Unit1.Em7.ControlNodes".cm.softCam.sepaGripperAxisZ.waitPos.inPos;
   #statTonTime[180].TON(IN := #_w1 AND "Unit1.Em7.ControlNodes".sepaGripper."step".transition1[180],
                         PT := T#1000ms);
   IF #statTonTime[180].Q THEN
       "Unit1.Em7.ControlNodes".sepaGripper.sequence.status.nextStep := #JOB_1_STEP_90;
   END_IF;
END_REGION

REGION Network 15: Step[190] : Job[1] Step End
   RUNG wire#powerrail
      { S7_Templates := "SrcType := DInt" } EQ_Contact(in1 := "Unit1.Em7.ControlNodes".sepaGripper.sequence.status.currentStep, in2 := #JOB_1_STEP_90)
      Contact( "Unit1.Em7.ControlNodes".sepaGripper.sequence.status.seqActive )
      wire#w1
      Coil( "Unit1.Em7.ControlNodes".sepaGripper."step".action1[190] )
   END_RUNG
   RUNG wire#w1
      Coil( "Unit1.Em7.ControlNodes".sepaGripper."step".transition1[190] )
   END_RUNG
   RUNG wire#w1
      Contact( "Unit1.Em7.ControlNodes".sepaGripper."step".transition1[190] )
      { S7_Templates := "time_type := Time" } #statTonTime[190].TON(pt := T#1000ms, et =>)
      Move(in := #STEP_IDLE, out1 => "Unit1.Em7.ControlNodes".sepaGripper.sequence.status.nextStep)
   END_RUNG
   // the same network as SCL:
   "Unit1.Em7.ControlNodes".sepaGripper."step".action1[190] := ("Unit1.Em7.ControlNodes".sepaGripper.sequence.status.currentStep = #JOB_1_STEP_90) AND "Unit1.Em7.ControlNodes".sepaGripper.sequence.status.seqActive;
   "Unit1.Em7.ControlNodes".sepaGripper."step".transition1[190] := ("Unit1.Em7.ControlNodes".sepaGripper.sequence.status.currentStep = #JOB_1_STEP_90) AND "Unit1.Em7.ControlNodes".sepaGripper.sequence.status.seqActive;
   #statTonTime[190].TON(IN := ("Unit1.Em7.ControlNodes".sepaGripper.sequence.status.currentStep = #JOB_1_STEP_90) AND "Unit1.Em7.ControlNodes".sepaGripper.sequence.status.seqActive AND "Unit1.Em7.ControlNodes".sepaGripper."step".transition1[190],
                         PT := T#1000ms);
   IF #statTonTime[190].Q THEN
       "Unit1.Em7.ControlNodes".sepaGripper.sequence.status.nextStep := #STEP_IDLE;
   END_IF;
END_REGION

REGION Network 16: ******************** JOB[2] Load ********************
END_REGION

REGION Network 17: Step[201] : JOB[2] Condition
   RUNG wire#powerrail
      { S7_Templates := "SrcType := DInt" } EQ_Contact(in1 := "Unit1.Em7.ControlNodes".sepaGripper.sequence.status.currentStep, in2 := #JOB_2_STEP_01)
      Contact( "Unit1.Em7.ControlNodes".sepaGripper.sequence.status.seqActive )
      wire#w1
      Coil( "Unit1.Em7.ControlNodes".sepaGripper."step".action1[201] )
   END_RUNG
   RUNG wire#w1
      Coil( "Unit1.Em7.ControlNodes".sepaGripper."step".transition1[201] )
   END_RUNG
   RUNG wire#w1
      Contact( "Unit1.Em7.ControlNodes".sepaGripper."step".transition1[201] )
      { S7_Templates := "time_type := Time" } #statTonTime[201].TON(pt := T#1000ms, et =>)
      Move(in := #JOB_2_STEP_10, out1 => "Unit1.Em7.ControlNodes".sepaGripper.sequence.status.nextStep)
   END_RUNG
   // the same network as SCL:
   "Unit1.Em7.ControlNodes".sepaGripper."step".action1[201] := ("Unit1.Em7.ControlNodes".sepaGripper.sequence.status.currentStep = #JOB_2_STEP_01) AND "Unit1.Em7.ControlNodes".sepaGripper.sequence.status.seqActive;
   "Unit1.Em7.ControlNodes".sepaGripper."step".transition1[201] := ("Unit1.Em7.ControlNodes".sepaGripper.sequence.status.currentStep = #JOB_2_STEP_01) AND "Unit1.Em7.ControlNodes".sepaGripper.sequence.status.seqActive;
   #statTonTime[201].TON(IN := ("Unit1.Em7.ControlNodes".sepaGripper.sequence.status.currentStep = #JOB_2_STEP_01) AND "Unit1.Em7.ControlNodes".sepaGripper.sequence.status.seqActive AND "Unit1.Em7.ControlNodes".sepaGripper."step".transition1[201],
                         PT := T#1000ms);
   IF #statTonTime[201].Q THEN
       "Unit1.Em7.ControlNodes".sepaGripper.sequence.status.nextStep := #JOB_2_STEP_10;
   END_IF;
END_REGION

REGION Network 18: Step[210] : Gripper X,Z-Axis Load Pos
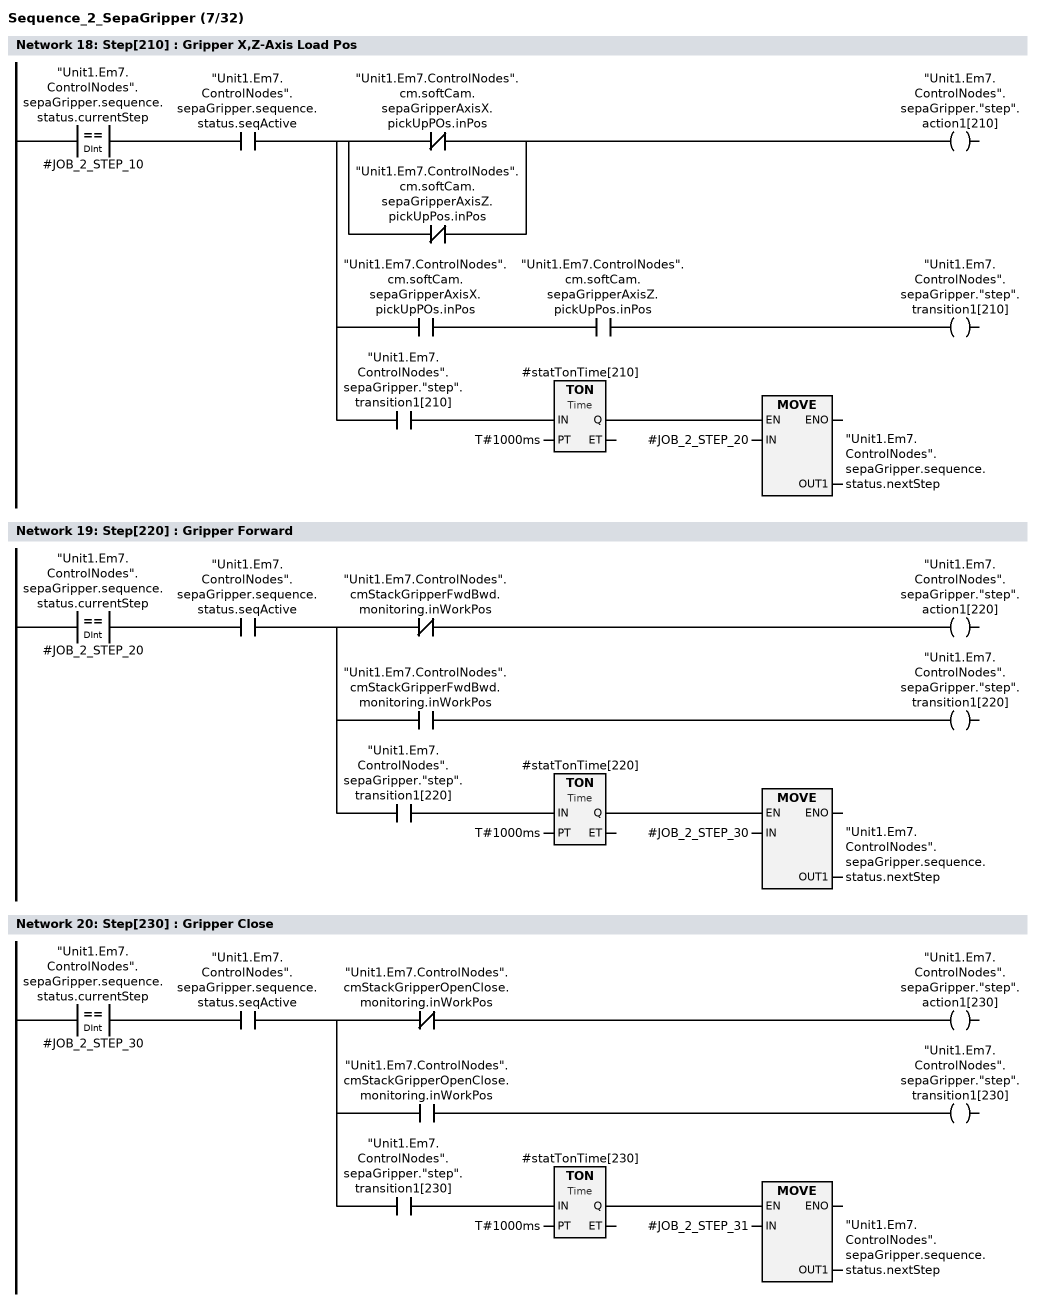
   RUNG wire#powerrail
      { S7_Templates := "SrcType := DInt" } EQ_Contact(in1 := "Unit1.Em7.ControlNodes".sepaGripper.sequence.status.currentStep, in2 := #JOB_2_STEP_10)
      Contact( "Unit1.Em7.ControlNodes".sepaGripper.sequence.status.seqActive )
      wire#w1
      I_Contact( "Unit1.Em7.ControlNodes".cm.softCam.sepaGripperAxisX.pickUpPOs.inPos )
      wire#w2
      Coil( "Unit1.Em7.ControlNodes".sepaGripper."step".action1[210] )
   END_RUNG
   RUNG wire#w1
      I_Contact( "Unit1.Em7.ControlNodes".cm.softCam.sepaGripperAxisZ.pickUpPos.inPos )
   END_RUNG wire#w2
   RUNG wire#w1
      Contact( "Unit1.Em7.ControlNodes".cm.softCam.sepaGripperAxisX.pickUpPOs.inPos )
      Contact( "Unit1.Em7.ControlNodes".cm.softCam.sepaGripperAxisZ.pickUpPos.inPos )
      Coil( "Unit1.Em7.ControlNodes".sepaGripper."step".transition1[210] )
   END_RUNG
   RUNG wire#w1
      Contact( "Unit1.Em7.ControlNodes".sepaGripper."step".transition1[210] )
      { S7_Templates := "time_type := Time" } #statTonTime[210].TON(pt := T#1000ms, et =>)
      Move(in := #JOB_2_STEP_20, out1 => "Unit1.Em7.ControlNodes".sepaGripper.sequence.status.nextStep)
   END_RUNG
   // the same network as SCL:
   #_w1 := ("Unit1.Em7.ControlNodes".sepaGripper.sequence.status.currentStep = #JOB_2_STEP_10) AND "Unit1.Em7.ControlNodes".sepaGripper.sequence.status.seqActive;
   "Unit1.Em7.ControlNodes".sepaGripper."step".action1[210] := #_w1 AND (NOT "Unit1.Em7.ControlNodes".cm.softCam.sepaGripperAxisX.pickUpPOs.inPos OR NOT "Unit1.Em7.ControlNodes".cm.softCam.sepaGripperAxisZ.pickUpPos.inPos);
   "Unit1.Em7.ControlNodes".sepaGripper."step".transition1[210] := #_w1 AND "Unit1.Em7.ControlNodes".cm.softCam.sepaGripperAxisX.pickUpPOs.inPos AND "Unit1.Em7.ControlNodes".cm.softCam.sepaGripperAxisZ.pickUpPos.inPos;
   #statTonTime[210].TON(IN := #_w1 AND "Unit1.Em7.ControlNodes".sepaGripper."step".transition1[210],
                         PT := T#1000ms);
   IF #statTonTime[210].Q THEN
       "Unit1.Em7.ControlNodes".sepaGripper.sequence.status.nextStep := #JOB_2_STEP_20;
   END_IF;
END_REGION

REGION Network 19: Step[220] : Gripper Forward
   RUNG wire#powerrail
      { S7_Templates := "SrcType := DInt" } EQ_Contact(in1 := "Unit1.Em7.ControlNodes".sepaGripper.sequence.status.currentStep, in2 := #JOB_2_STEP_20)
      Contact( "Unit1.Em7.ControlNodes".sepaGripper.sequence.status.seqActive )
      wire#w1
      I_Contact( "Unit1.Em7.ControlNodes".cmStackGripperFwdBwd.monitoring.inWorkPos )
      Coil( "Unit1.Em7.ControlNodes".sepaGripper."step".action1[220] )
   END_RUNG
   RUNG wire#w1
      Contact( "Unit1.Em7.ControlNodes".cmStackGripperFwdBwd.monitoring.inWorkPos )
      Coil( "Unit1.Em7.ControlNodes".sepaGripper."step".transition1[220] )
   END_RUNG
   RUNG wire#w1
      Contact( "Unit1.Em7.ControlNodes".sepaGripper."step".transition1[220] )
      { S7_Templates := "time_type := Time" } #statTonTime[220].TON(pt := T#1000ms, et =>)
      Move(in := #JOB_2_STEP_30, out1 => "Unit1.Em7.ControlNodes".sepaGripper.sequence.status.nextStep)
   END_RUNG
   // the same network as SCL:
   #_w1 := ("Unit1.Em7.ControlNodes".sepaGripper.sequence.status.currentStep = #JOB_2_STEP_20) AND "Unit1.Em7.ControlNodes".sepaGripper.sequence.status.seqActive;
   "Unit1.Em7.ControlNodes".sepaGripper."step".action1[220] := #_w1 AND NOT "Unit1.Em7.ControlNodes".cmStackGripperFwdBwd.monitoring.inWorkPos;
   "Unit1.Em7.ControlNodes".sepaGripper."step".transition1[220] := #_w1 AND "Unit1.Em7.ControlNodes".cmStackGripperFwdBwd.monitoring.inWorkPos;
   #statTonTime[220].TON(IN := #_w1 AND "Unit1.Em7.ControlNodes".sepaGripper."step".transition1[220],
                         PT := T#1000ms);
   IF #statTonTime[220].Q THEN
       "Unit1.Em7.ControlNodes".sepaGripper.sequence.status.nextStep := #JOB_2_STEP_30;
   END_IF;
END_REGION

REGION Network 20: Step[230] : Gripper Close
   RUNG wire#powerrail
      { S7_Templates := "SrcType := DInt" } EQ_Contact(in1 := "Unit1.Em7.ControlNodes".sepaGripper.sequence.status.currentStep, in2 := #JOB_2_STEP_30)
      Contact( "Unit1.Em7.ControlNodes".sepaGripper.sequence.status.seqActive )
      wire#w1
      I_Contact( "Unit1.Em7.ControlNodes".cmStackGripperOpenClose.monitoring.inWorkPos )
      Coil( "Unit1.Em7.ControlNodes".sepaGripper."step".action1[230] )
   END_RUNG
   RUNG wire#w1
      Contact( "Unit1.Em7.ControlNodes".cmStackGripperOpenClose.monitoring.inWorkPos )
      Coil( "Unit1.Em7.ControlNodes".sepaGripper."step".transition1[230] )
   END_RUNG
   RUNG wire#w1
      Contact( "Unit1.Em7.ControlNodes".sepaGripper."step".transition1[230] )
      { S7_Templates := "time_type := Time" } #statTonTime[230].TON(pt := T#1000ms, et =>)
      Move(in := #JOB_2_STEP_31, out1 => "Unit1.Em7.ControlNodes".sepaGripper.sequence.status.nextStep)
   END_RUNG
   // the same network as SCL:
   #_w1 := ("Unit1.Em7.ControlNodes".sepaGripper.sequence.status.currentStep = #JOB_2_STEP_30) AND "Unit1.Em7.ControlNodes".sepaGripper.sequence.status.seqActive;
   "Unit1.Em7.ControlNodes".sepaGripper."step".action1[230] := #_w1 AND NOT "Unit1.Em7.ControlNodes".cmStackGripperOpenClose.monitoring.inWorkPos;
   "Unit1.Em7.ControlNodes".sepaGripper."step".transition1[230] := #_w1 AND "Unit1.Em7.ControlNodes".cmStackGripperOpenClose.monitoring.inWorkPos;
   #statTonTime[230].TON(IN := #_w1 AND "Unit1.Em7.ControlNodes".sepaGripper."step".transition1[230],
                         PT := T#1000ms);
   IF #statTonTime[230].Q THEN
       "Unit1.Em7.ControlNodes".sepaGripper.sequence.status.nextStep := #JOB_2_STEP_31;
   END_IF;
END_REGION

REGION Network 21: Step[231] : Sepa Gripper → Stack Table [Loading Ready]
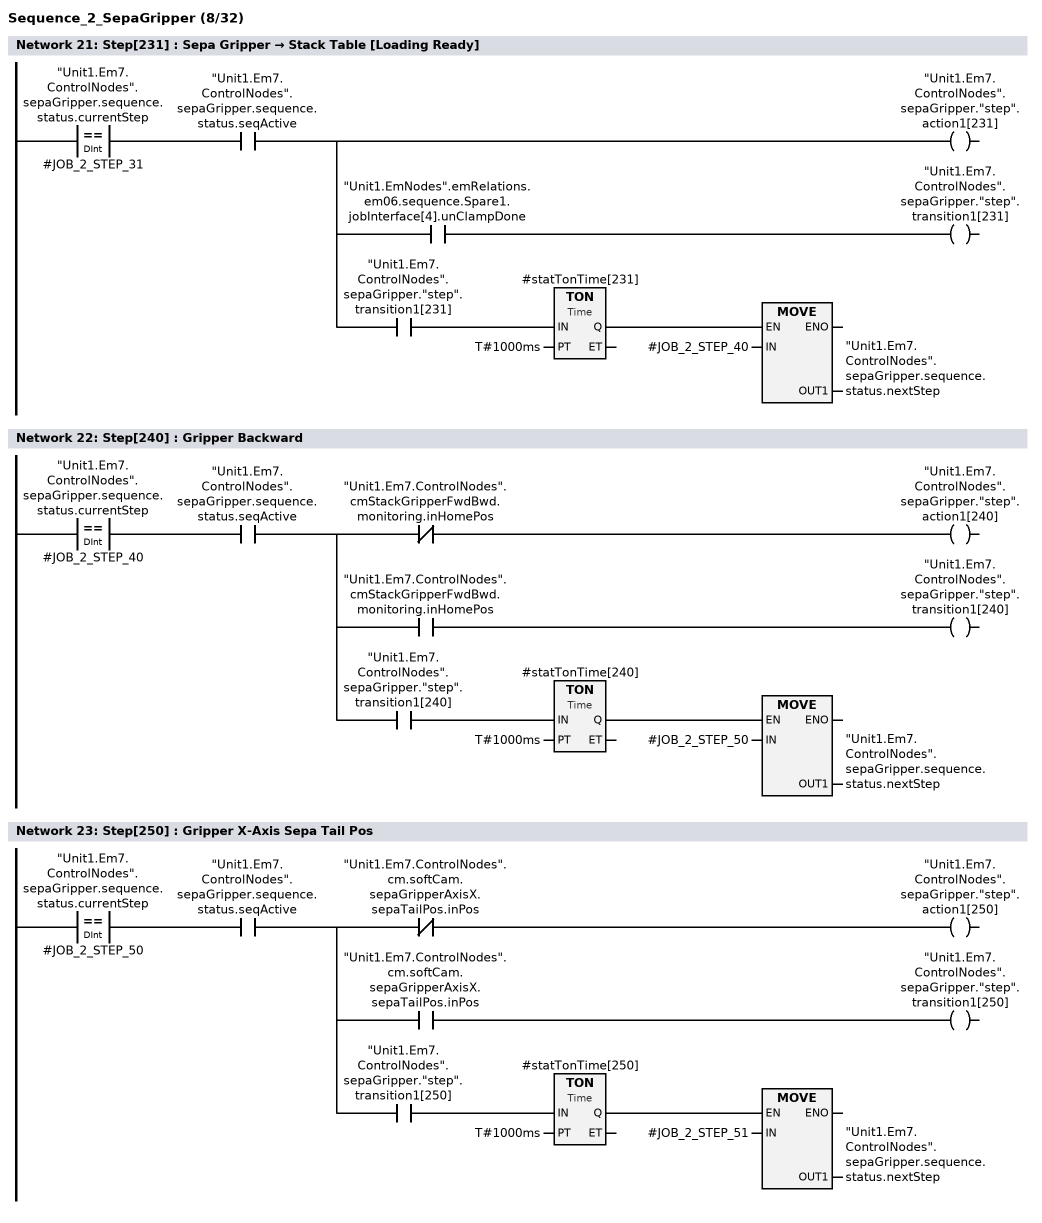
   RUNG wire#powerrail
      { S7_Templates := "SrcType := DInt" } EQ_Contact(in1 := "Unit1.Em7.ControlNodes".sepaGripper.sequence.status.currentStep, in2 := #JOB_2_STEP_31)
      Contact( "Unit1.Em7.ControlNodes".sepaGripper.sequence.status.seqActive )
      wire#w1
      Coil( "Unit1.Em7.ControlNodes".sepaGripper."step".action1[231] )
   END_RUNG
   RUNG wire#w1
      Contact( "Unit1.EmNodes".emRelations.em06.sequence.Spare1.jobInterface[4].unClampDone )
      Coil( "Unit1.Em7.ControlNodes".sepaGripper."step".transition1[231] )
   END_RUNG
   RUNG wire#w1
      Contact( "Unit1.Em7.ControlNodes".sepaGripper."step".transition1[231] )
      { S7_Templates := "time_type := Time" } #statTonTime[231].TON(pt := T#1000ms, et =>)
      Move(in := #JOB_2_STEP_40, out1 => "Unit1.Em7.ControlNodes".sepaGripper.sequence.status.nextStep)
   END_RUNG
   // the same network as SCL:
   "Unit1.Em7.ControlNodes".sepaGripper."step".action1[231] := ("Unit1.Em7.ControlNodes".sepaGripper.sequence.status.currentStep = #JOB_2_STEP_31) AND "Unit1.Em7.ControlNodes".sepaGripper.sequence.status.seqActive;
   "Unit1.Em7.ControlNodes".sepaGripper."step".transition1[231] := ("Unit1.Em7.ControlNodes".sepaGripper.sequence.status.currentStep = #JOB_2_STEP_31) AND "Unit1.Em7.ControlNodes".sepaGripper.sequence.status.seqActive AND "Unit1.EmNodes".emRelations.em06.sequence.Spare1.jobInterface[4].unClampDone;
   #statTonTime[231].TON(IN := ("Unit1.Em7.ControlNodes".sepaGripper.sequence.status.currentStep = #JOB_2_STEP_31) AND "Unit1.Em7.ControlNodes".sepaGripper.sequence.status.seqActive AND "Unit1.Em7.ControlNodes".sepaGripper."step".transition1[231],
                         PT := T#1000ms);
   IF #statTonTime[231].Q THEN
       "Unit1.Em7.ControlNodes".sepaGripper.sequence.status.nextStep := #JOB_2_STEP_40;
   END_IF;
END_REGION

REGION Network 22: Step[240] : Gripper Backward
   RUNG wire#powerrail
      { S7_Templates := "SrcType := DInt" } EQ_Contact(in1 := "Unit1.Em7.ControlNodes".sepaGripper.sequence.status.currentStep, in2 := #JOB_2_STEP_40)
      Contact( "Unit1.Em7.ControlNodes".sepaGripper.sequence.status.seqActive )
      wire#w1
      I_Contact( "Unit1.Em7.ControlNodes".cmStackGripperFwdBwd.monitoring.inHomePos )
      Coil( "Unit1.Em7.ControlNodes".sepaGripper."step".action1[240] )
   END_RUNG
   RUNG wire#w1
      Contact( "Unit1.Em7.ControlNodes".cmStackGripperFwdBwd.monitoring.inHomePos )
      Coil( "Unit1.Em7.ControlNodes".sepaGripper."step".transition1[240] )
   END_RUNG
   RUNG wire#w1
      Contact( "Unit1.Em7.ControlNodes".sepaGripper."step".transition1[240] )
      { S7_Templates := "time_type := Time" } #statTonTime[240].TON(pt := T#1000ms, et =>)
      Move(in := #JOB_2_STEP_50, out1 => "Unit1.Em7.ControlNodes".sepaGripper.sequence.status.nextStep)
   END_RUNG
   // the same network as SCL:
   #_w1 := ("Unit1.Em7.ControlNodes".sepaGripper.sequence.status.currentStep = #JOB_2_STEP_40) AND "Unit1.Em7.ControlNodes".sepaGripper.sequence.status.seqActive;
   "Unit1.Em7.ControlNodes".sepaGripper."step".action1[240] := #_w1 AND NOT "Unit1.Em7.ControlNodes".cmStackGripperFwdBwd.monitoring.inHomePos;
   "Unit1.Em7.ControlNodes".sepaGripper."step".transition1[240] := #_w1 AND "Unit1.Em7.ControlNodes".cmStackGripperFwdBwd.monitoring.inHomePos;
   #statTonTime[240].TON(IN := #_w1 AND "Unit1.Em7.ControlNodes".sepaGripper."step".transition1[240],
                         PT := T#1000ms);
   IF #statTonTime[240].Q THEN
       "Unit1.Em7.ControlNodes".sepaGripper.sequence.status.nextStep := #JOB_2_STEP_50;
   END_IF;
END_REGION

REGION Network 23: Step[250] : Gripper X-Axis Sepa Tail Pos
   RUNG wire#powerrail
      { S7_Templates := "SrcType := DInt" } EQ_Contact(in1 := "Unit1.Em7.ControlNodes".sepaGripper.sequence.status.currentStep, in2 := #JOB_2_STEP_50)
      Contact( "Unit1.Em7.ControlNodes".sepaGripper.sequence.status.seqActive )
      wire#w1
      I_Contact( "Unit1.Em7.ControlNodes".cm.softCam.sepaGripperAxisX.sepaTailPos.inPos )
      Coil( "Unit1.Em7.ControlNodes".sepaGripper."step".action1[250] )
   END_RUNG
   RUNG wire#w1
      Contact( "Unit1.Em7.ControlNodes".cm.softCam.sepaGripperAxisX.sepaTailPos.inPos )
      Coil( "Unit1.Em7.ControlNodes".sepaGripper."step".transition1[250] )
   END_RUNG
   RUNG wire#w1
      Contact( "Unit1.Em7.ControlNodes".sepaGripper."step".transition1[250] )
      { S7_Templates := "time_type := Time" } #statTonTime[250].TON(pt := T#1000ms, et =>)
      Move(in := #JOB_2_STEP_51, out1 => "Unit1.Em7.ControlNodes".sepaGripper.sequence.status.nextStep)
   END_RUNG
   // the same network as SCL:
   #_w1 := ("Unit1.Em7.ControlNodes".sepaGripper.sequence.status.currentStep = #JOB_2_STEP_50) AND "Unit1.Em7.ControlNodes".sepaGripper.sequence.status.seqActive;
   "Unit1.Em7.ControlNodes".sepaGripper."step".action1[250] := #_w1 AND NOT "Unit1.Em7.ControlNodes".cm.softCam.sepaGripperAxisX.sepaTailPos.inPos;
   "Unit1.Em7.ControlNodes".sepaGripper."step".transition1[250] := #_w1 AND "Unit1.Em7.ControlNodes".cm.softCam.sepaGripperAxisX.sepaTailPos.inPos;
   #statTonTime[250].TON(IN := #_w1 AND "Unit1.Em7.ControlNodes".sepaGripper."step".transition1[250],
                         PT := T#1000ms);
   IF #statTonTime[250].Q THEN
       "Unit1.Em7.ControlNodes".sepaGripper.sequence.status.nextStep := #JOB_2_STEP_51;
   END_IF;
END_REGION

REGION Network 24: Step[251] : Gripper → Stack Table [Loading Done]
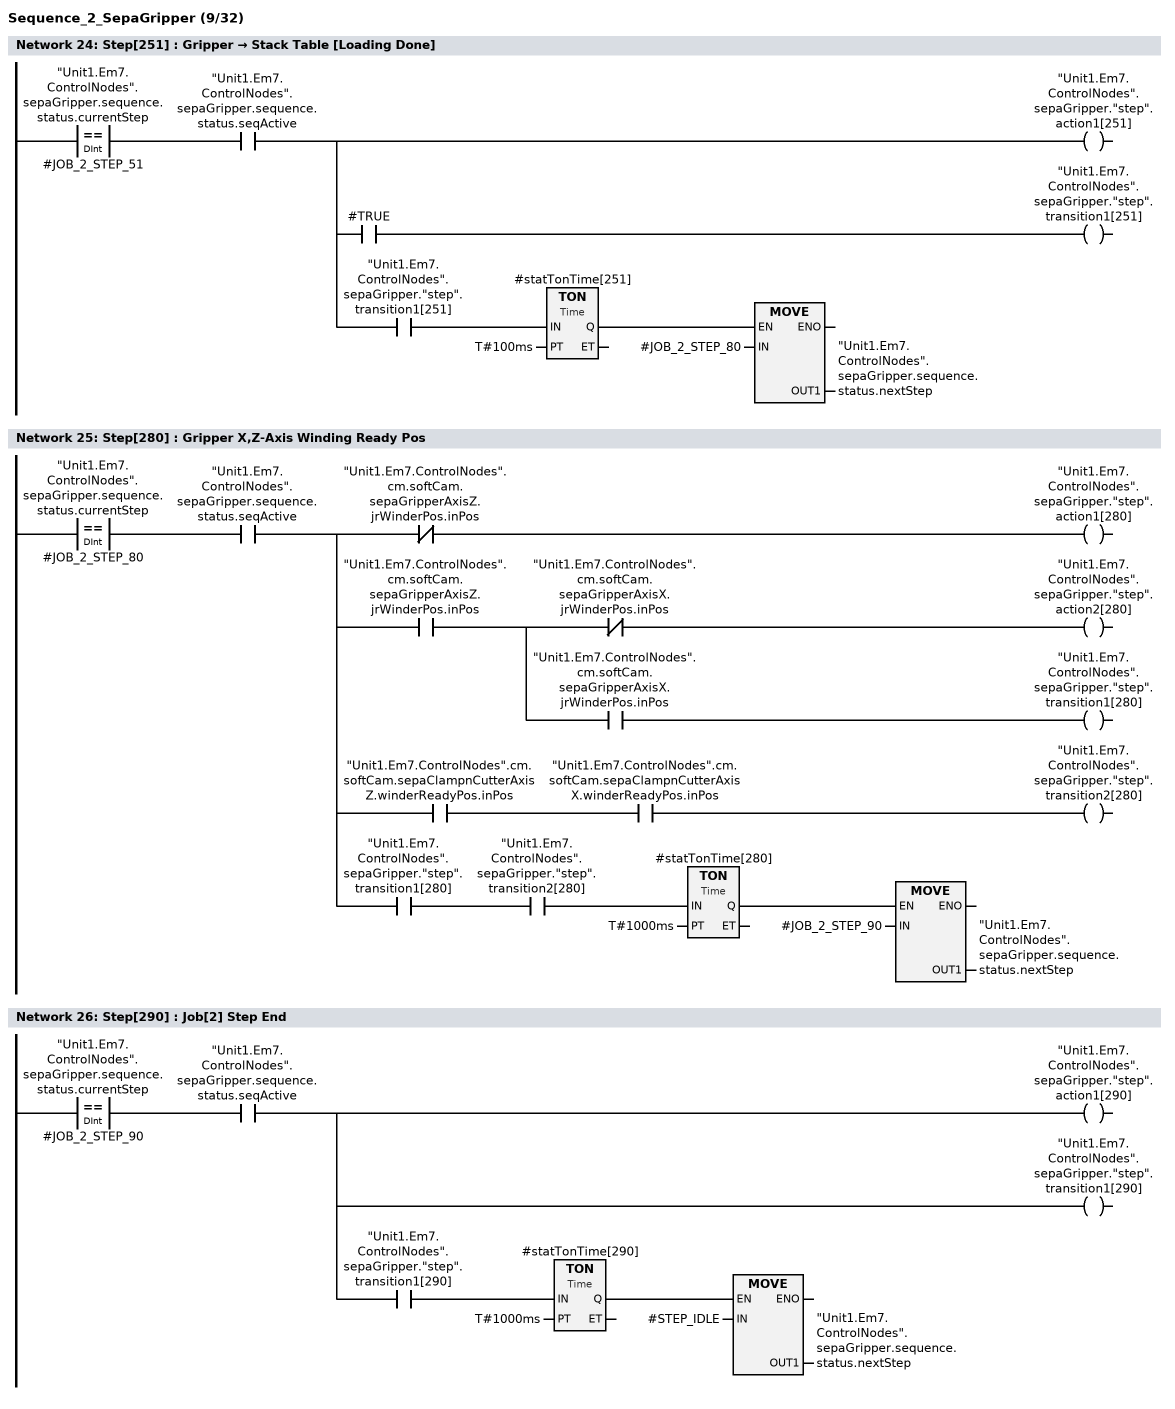
   RUNG wire#powerrail
      { S7_Templates := "SrcType := DInt" } EQ_Contact(in1 := "Unit1.Em7.ControlNodes".sepaGripper.sequence.status.currentStep, in2 := #JOB_2_STEP_51)
      Contact( "Unit1.Em7.ControlNodes".sepaGripper.sequence.status.seqActive )
      wire#w1
      Coil( "Unit1.Em7.ControlNodes".sepaGripper."step".action1[251] )
   END_RUNG
   RUNG wire#w1
      Contact( #TRUE )
      Coil( "Unit1.Em7.ControlNodes".sepaGripper."step".transition1[251] )
   END_RUNG
   RUNG wire#w1
      Contact( "Unit1.Em7.ControlNodes".sepaGripper."step".transition1[251] )
      { S7_Templates := "time_type := Time" } #statTonTime[251].TON(pt := T#100ms, et =>)
      Move(in := #JOB_2_STEP_80, out1 => "Unit1.Em7.ControlNodes".sepaGripper.sequence.status.nextStep)
   END_RUNG
   // the same network as SCL:
   "Unit1.Em7.ControlNodes".sepaGripper."step".action1[251] := ("Unit1.Em7.ControlNodes".sepaGripper.sequence.status.currentStep = #JOB_2_STEP_51) AND "Unit1.Em7.ControlNodes".sepaGripper.sequence.status.seqActive;
   "Unit1.Em7.ControlNodes".sepaGripper."step".transition1[251] := ("Unit1.Em7.ControlNodes".sepaGripper.sequence.status.currentStep = #JOB_2_STEP_51) AND "Unit1.Em7.ControlNodes".sepaGripper.sequence.status.seqActive AND #TRUE;
   #statTonTime[251].TON(IN := ("Unit1.Em7.ControlNodes".sepaGripper.sequence.status.currentStep = #JOB_2_STEP_51) AND "Unit1.Em7.ControlNodes".sepaGripper.sequence.status.seqActive AND "Unit1.Em7.ControlNodes".sepaGripper."step".transition1[251],
                         PT := T#100ms);
   IF #statTonTime[251].Q THEN
       "Unit1.Em7.ControlNodes".sepaGripper.sequence.status.nextStep := #JOB_2_STEP_80;
   END_IF;
END_REGION

REGION Network 25: Step[280] : Gripper X,Z-Axis Winding Ready Pos
   RUNG wire#powerrail
      { S7_Templates := "SrcType := DInt" } EQ_Contact(in1 := "Unit1.Em7.ControlNodes".sepaGripper.sequence.status.currentStep, in2 := #JOB_2_STEP_80)
      Contact( "Unit1.Em7.ControlNodes".sepaGripper.sequence.status.seqActive )
      wire#w1
      I_Contact( "Unit1.Em7.ControlNodes".cm.softCam.sepaGripperAxisZ.jrWinderPos.inPos )
      Coil( "Unit1.Em7.ControlNodes".sepaGripper."step".action1[280] )
   END_RUNG
   RUNG wire#w1
      Contact( "Unit1.Em7.ControlNodes".cm.softCam.sepaGripperAxisZ.jrWinderPos.inPos )
      wire#w2
      I_Contact( "Unit1.Em7.ControlNodes".cm.softCam.sepaGripperAxisX.jrWinderPos.inPos )
      Coil( "Unit1.Em7.ControlNodes".sepaGripper."step".action2[280] )
   END_RUNG
   RUNG wire#w2
      Contact( "Unit1.Em7.ControlNodes".cm.softCam.sepaGripperAxisX.jrWinderPos.inPos )
      Coil( "Unit1.Em7.ControlNodes".sepaGripper."step".transition1[280] )
   END_RUNG
   RUNG wire#w1
      Contact( "Unit1.Em7.ControlNodes".cm.softCam.sepaClampnCutterAxisZ.winderReadyPos.inPos )
      Contact( "Unit1.Em7.ControlNodes".cm.softCam.sepaClampnCutterAxisX.winderReadyPos.inPos )
      Coil( "Unit1.Em7.ControlNodes".sepaGripper."step".transition2[280] )
   END_RUNG
   RUNG wire#w1
      Contact( "Unit1.Em7.ControlNodes".sepaGripper."step".transition1[280] )
      Contact( "Unit1.Em7.ControlNodes".sepaGripper."step".transition2[280] )
      { S7_Templates := "time_type := Time" } #statTonTime[280].TON(pt := T#1000ms, et =>)
      Move(in := #JOB_2_STEP_90, out1 => "Unit1.Em7.ControlNodes".sepaGripper.sequence.status.nextStep)
   END_RUNG
   // the same network as SCL:
   #_w1 := ("Unit1.Em7.ControlNodes".sepaGripper.sequence.status.currentStep = #JOB_2_STEP_80) AND "Unit1.Em7.ControlNodes".sepaGripper.sequence.status.seqActive;
   "Unit1.Em7.ControlNodes".sepaGripper."step".action1[280] := #_w1 AND NOT "Unit1.Em7.ControlNodes".cm.softCam.sepaGripperAxisZ.jrWinderPos.inPos;
   #_w2 := #_w1 AND "Unit1.Em7.ControlNodes".cm.softCam.sepaGripperAxisZ.jrWinderPos.inPos;
   "Unit1.Em7.ControlNodes".sepaGripper."step".action2[280] := #_w2 AND NOT "Unit1.Em7.ControlNodes".cm.softCam.sepaGripperAxisX.jrWinderPos.inPos;
   "Unit1.Em7.ControlNodes".sepaGripper."step".transition1[280] := #_w2 AND "Unit1.Em7.ControlNodes".cm.softCam.sepaGripperAxisX.jrWinderPos.inPos;
   "Unit1.Em7.ControlNodes".sepaGripper."step".transition2[280] := #_w1 AND "Unit1.Em7.ControlNodes".cm.softCam.sepaClampnCutterAxisZ.winderReadyPos.inPos AND "Unit1.Em7.ControlNodes".cm.softCam.sepaClampnCutterAxisX.winderReadyPos.inPos;
   #statTonTime[280].TON(IN := #_w1 AND "Unit1.Em7.ControlNodes".sepaGripper."step".transition1[280] AND "Unit1.Em7.ControlNodes".sepaGripper."step".transition2[280],
                         PT := T#1000ms);
   IF #statTonTime[280].Q THEN
       "Unit1.Em7.ControlNodes".sepaGripper.sequence.status.nextStep := #JOB_2_STEP_90;
   END_IF;
END_REGION

REGION Network 26: Step[290] : Job[2] Step End
   RUNG wire#powerrail
      { S7_Templates := "SrcType := DInt" } EQ_Contact(in1 := "Unit1.Em7.ControlNodes".sepaGripper.sequence.status.currentStep, in2 := #JOB_2_STEP_90)
      Contact( "Unit1.Em7.ControlNodes".sepaGripper.sequence.status.seqActive )
      wire#w1
      Coil( "Unit1.Em7.ControlNodes".sepaGripper."step".action1[290] )
   END_RUNG
   RUNG wire#w1
      Coil( "Unit1.Em7.ControlNodes".sepaGripper."step".transition1[290] )
   END_RUNG
   RUNG wire#w1
      Contact( "Unit1.Em7.ControlNodes".sepaGripper."step".transition1[290] )
      { S7_Templates := "time_type := Time" } #statTonTime[290].TON(pt := T#1000ms, et =>)
      Move(in := #STEP_IDLE, out1 => "Unit1.Em7.ControlNodes".sepaGripper.sequence.status.nextStep)
   END_RUNG
   // the same network as SCL:
   "Unit1.Em7.ControlNodes".sepaGripper."step".action1[290] := ("Unit1.Em7.ControlNodes".sepaGripper.sequence.status.currentStep = #JOB_2_STEP_90) AND "Unit1.Em7.ControlNodes".sepaGripper.sequence.status.seqActive;
   "Unit1.Em7.ControlNodes".sepaGripper."step".transition1[290] := ("Unit1.Em7.ControlNodes".sepaGripper.sequence.status.currentStep = #JOB_2_STEP_90) AND "Unit1.Em7.ControlNodes".sepaGripper.sequence.status.seqActive;
   #statTonTime[290].TON(IN := ("Unit1.Em7.ControlNodes".sepaGripper.sequence.status.currentStep = #JOB_2_STEP_90) AND "Unit1.Em7.ControlNodes".sepaGripper.sequence.status.seqActive AND "Unit1.Em7.ControlNodes".sepaGripper."step".transition1[290],
                         PT := T#1000ms);
   IF #statTonTime[290].Q THEN
       "Unit1.Em7.ControlNodes".sepaGripper.sequence.status.nextStep := #STEP_IDLE;
   END_IF;
END_REGION

REGION Network 27: ******************** JOB[3] Unload ********************
END_REGION

REGION Network 28: Step[301] : JOB[3] Condition
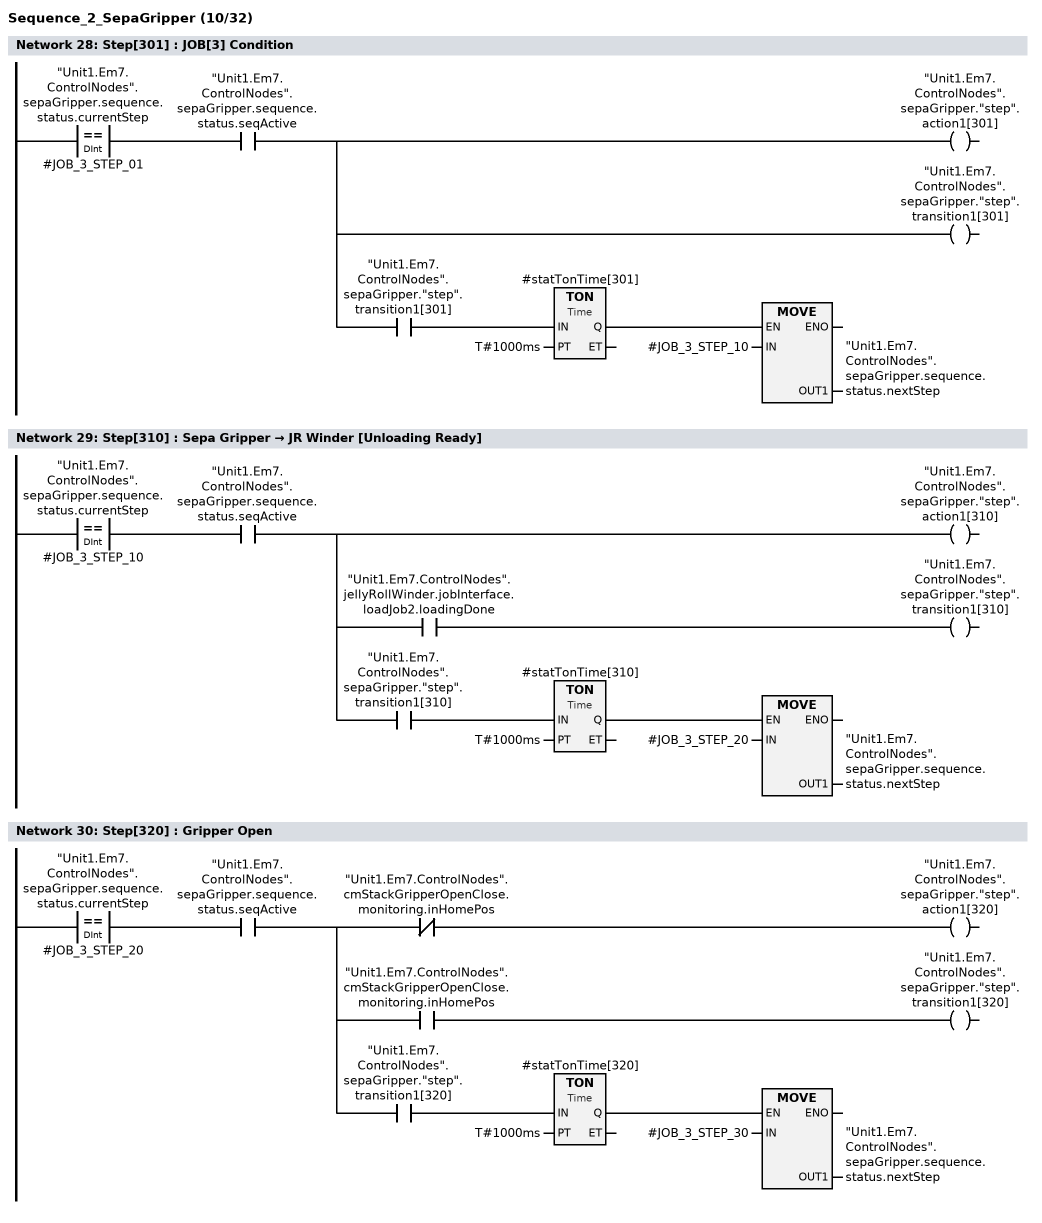
   RUNG wire#powerrail
      { S7_Templates := "SrcType := DInt" } EQ_Contact(in1 := "Unit1.Em7.ControlNodes".sepaGripper.sequence.status.currentStep, in2 := #JOB_3_STEP_01)
      Contact( "Unit1.Em7.ControlNodes".sepaGripper.sequence.status.seqActive )
      wire#w1
      Coil( "Unit1.Em7.ControlNodes".sepaGripper."step".action1[301] )
   END_RUNG
   RUNG wire#w1
      Coil( "Unit1.Em7.ControlNodes".sepaGripper."step".transition1[301] )
   END_RUNG
   RUNG wire#w1
      Contact( "Unit1.Em7.ControlNodes".sepaGripper."step".transition1[301] )
      { S7_Templates := "time_type := Time" } #statTonTime[301].TON(pt := T#1000ms, et =>)
      Move(in := #JOB_3_STEP_10, out1 => "Unit1.Em7.ControlNodes".sepaGripper.sequence.status.nextStep)
   END_RUNG
   // the same network as SCL:
   "Unit1.Em7.ControlNodes".sepaGripper."step".action1[301] := ("Unit1.Em7.ControlNodes".sepaGripper.sequence.status.currentStep = #JOB_3_STEP_01) AND "Unit1.Em7.ControlNodes".sepaGripper.sequence.status.seqActive;
   "Unit1.Em7.ControlNodes".sepaGripper."step".transition1[301] := ("Unit1.Em7.ControlNodes".sepaGripper.sequence.status.currentStep = #JOB_3_STEP_01) AND "Unit1.Em7.ControlNodes".sepaGripper.sequence.status.seqActive;
   #statTonTime[301].TON(IN := ("Unit1.Em7.ControlNodes".sepaGripper.sequence.status.currentStep = #JOB_3_STEP_01) AND "Unit1.Em7.ControlNodes".sepaGripper.sequence.status.seqActive AND "Unit1.Em7.ControlNodes".sepaGripper."step".transition1[301],
                         PT := T#1000ms);
   IF #statTonTime[301].Q THEN
       "Unit1.Em7.ControlNodes".sepaGripper.sequence.status.nextStep := #JOB_3_STEP_10;
   END_IF;
END_REGION

REGION Network 29: Step[310] : Sepa Gripper → JR Winder [Unloading Ready]
   RUNG wire#powerrail
      { S7_Templates := "SrcType := DInt" } EQ_Contact(in1 := "Unit1.Em7.ControlNodes".sepaGripper.sequence.status.currentStep, in2 := #JOB_3_STEP_10)
      Contact( "Unit1.Em7.ControlNodes".sepaGripper.sequence.status.seqActive )
      wire#w1
      Coil( "Unit1.Em7.ControlNodes".sepaGripper."step".action1[310] )
   END_RUNG
   RUNG wire#w1
      Contact( "Unit1.Em7.ControlNodes".jellyRollWinder.jobInterface.loadJob2.loadingDone )
      Coil( "Unit1.Em7.ControlNodes".sepaGripper."step".transition1[310] )
   END_RUNG
   RUNG wire#w1
      Contact( "Unit1.Em7.ControlNodes".sepaGripper."step".transition1[310] )
      { S7_Templates := "time_type := Time" } #statTonTime[310].TON(pt := T#1000ms, et =>)
      Move(in := #JOB_3_STEP_20, out1 => "Unit1.Em7.ControlNodes".sepaGripper.sequence.status.nextStep)
   END_RUNG
   // the same network as SCL:
   "Unit1.Em7.ControlNodes".sepaGripper."step".action1[310] := ("Unit1.Em7.ControlNodes".sepaGripper.sequence.status.currentStep = #JOB_3_STEP_10) AND "Unit1.Em7.ControlNodes".sepaGripper.sequence.status.seqActive;
   "Unit1.Em7.ControlNodes".sepaGripper."step".transition1[310] := ("Unit1.Em7.ControlNodes".sepaGripper.sequence.status.currentStep = #JOB_3_STEP_10) AND "Unit1.Em7.ControlNodes".sepaGripper.sequence.status.seqActive AND "Unit1.Em7.ControlNodes".jellyRollWinder.jobInterface.loadJob2.loadingDone;
   #statTonTime[310].TON(IN := ("Unit1.Em7.ControlNodes".sepaGripper.sequence.status.currentStep = #JOB_3_STEP_10) AND "Unit1.Em7.ControlNodes".sepaGripper.sequence.status.seqActive AND "Unit1.Em7.ControlNodes".sepaGripper."step".transition1[310],
                         PT := T#1000ms);
   IF #statTonTime[310].Q THEN
       "Unit1.Em7.ControlNodes".sepaGripper.sequence.status.nextStep := #JOB_3_STEP_20;
   END_IF;
END_REGION

REGION Network 30: Step[320] : Gripper Open
   RUNG wire#powerrail
      { S7_Templates := "SrcType := DInt" } EQ_Contact(in1 := "Unit1.Em7.ControlNodes".sepaGripper.sequence.status.currentStep, in2 := #JOB_3_STEP_20)
      Contact( "Unit1.Em7.ControlNodes".sepaGripper.sequence.status.seqActive )
      wire#w1
      I_Contact( "Unit1.Em7.ControlNodes".cmStackGripperOpenClose.monitoring.inHomePos )
      Coil( "Unit1.Em7.ControlNodes".sepaGripper."step".action1[320] )
   END_RUNG
   RUNG wire#w1
      Contact( "Unit1.Em7.ControlNodes".cmStackGripperOpenClose.monitoring.inHomePos )
      Coil( "Unit1.Em7.ControlNodes".sepaGripper."step".transition1[320] )
   END_RUNG
   RUNG wire#w1
      Contact( "Unit1.Em7.ControlNodes".sepaGripper."step".transition1[320] )
      { S7_Templates := "time_type := Time" } #statTonTime[320].TON(pt := T#1000ms, et =>)
      Move(in := #JOB_3_STEP_30, out1 => "Unit1.Em7.ControlNodes".sepaGripper.sequence.status.nextStep)
   END_RUNG
   // the same network as SCL:
   #_w1 := ("Unit1.Em7.ControlNodes".sepaGripper.sequence.status.currentStep = #JOB_3_STEP_20) AND "Unit1.Em7.ControlNodes".sepaGripper.sequence.status.seqActive;
   "Unit1.Em7.ControlNodes".sepaGripper."step".action1[320] := #_w1 AND NOT "Unit1.Em7.ControlNodes".cmStackGripperOpenClose.monitoring.inHomePos;
   "Unit1.Em7.ControlNodes".sepaGripper."step".transition1[320] := #_w1 AND "Unit1.Em7.ControlNodes".cmStackGripperOpenClose.monitoring.inHomePos;
   #statTonTime[320].TON(IN := #_w1 AND "Unit1.Em7.ControlNodes".sepaGripper."step".transition1[320],
                         PT := T#1000ms);
   IF #statTonTime[320].Q THEN
       "Unit1.Em7.ControlNodes".sepaGripper.sequence.status.nextStep := #JOB_3_STEP_30;
   END_IF;
END_REGION

REGION Network 31: Step[330] : Gripper X-Axis Avoid Pos
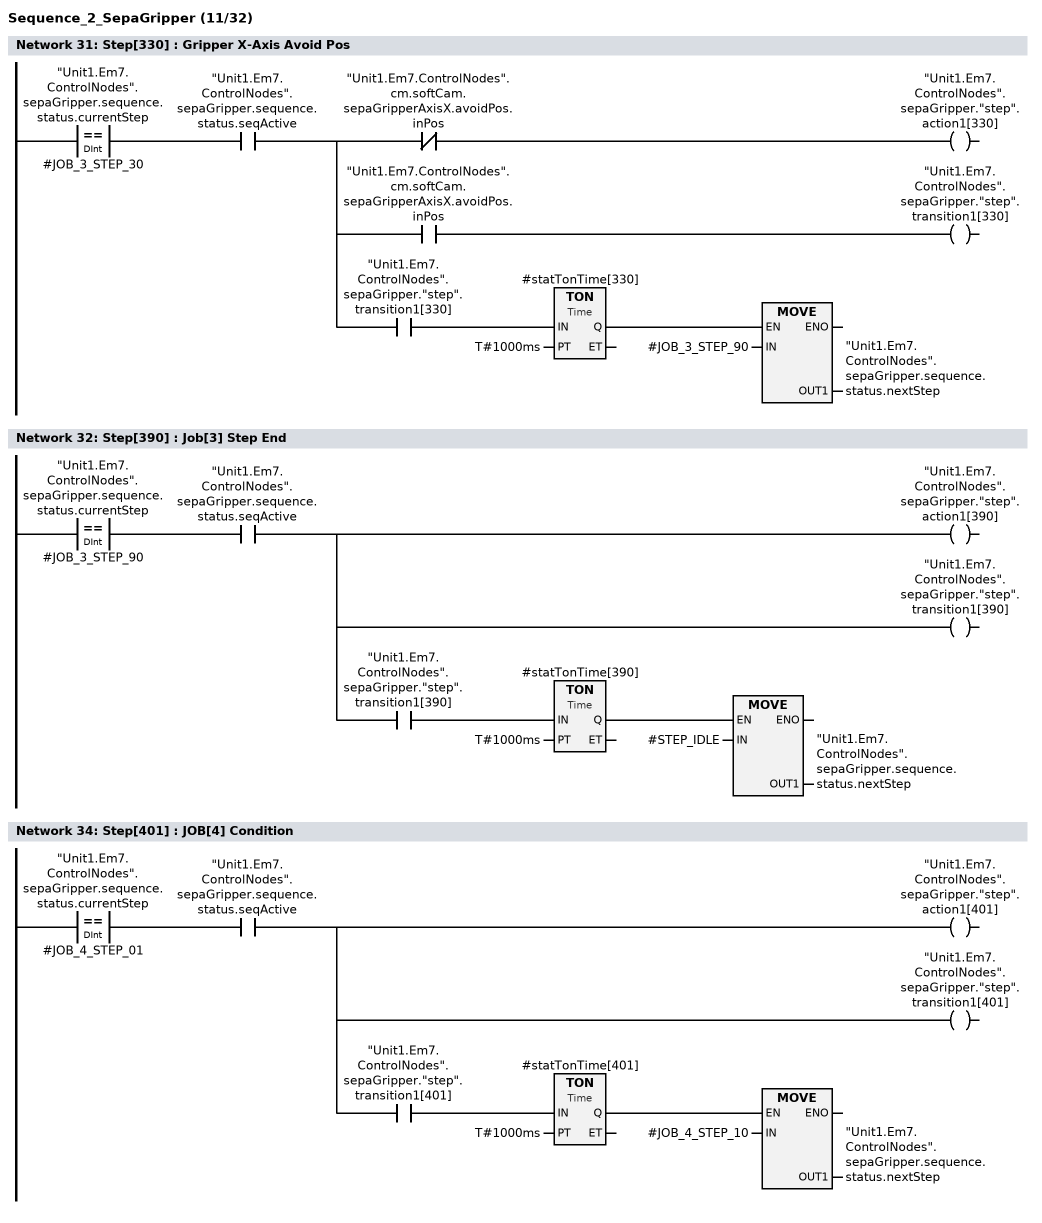
   RUNG wire#powerrail
      { S7_Templates := "SrcType := DInt" } EQ_Contact(in1 := "Unit1.Em7.ControlNodes".sepaGripper.sequence.status.currentStep, in2 := #JOB_3_STEP_30)
      Contact( "Unit1.Em7.ControlNodes".sepaGripper.sequence.status.seqActive )
      wire#w1
      I_Contact( "Unit1.Em7.ControlNodes".cm.softCam.sepaGripperAxisX.avoidPos.inPos )
      Coil( "Unit1.Em7.ControlNodes".sepaGripper."step".action1[330] )
   END_RUNG
   RUNG wire#w1
      Contact( "Unit1.Em7.ControlNodes".cm.softCam.sepaGripperAxisX.avoidPos.inPos )
      Coil( "Unit1.Em7.ControlNodes".sepaGripper."step".transition1[330] )
   END_RUNG
   RUNG wire#w1
      Contact( "Unit1.Em7.ControlNodes".sepaGripper."step".transition1[330] )
      { S7_Templates := "time_type := Time" } #statTonTime[330].TON(pt := T#1000ms, et =>)
      Move(in := #JOB_3_STEP_90, out1 => "Unit1.Em7.ControlNodes".sepaGripper.sequence.status.nextStep)
   END_RUNG
   // the same network as SCL:
   #_w1 := ("Unit1.Em7.ControlNodes".sepaGripper.sequence.status.currentStep = #JOB_3_STEP_30) AND "Unit1.Em7.ControlNodes".sepaGripper.sequence.status.seqActive;
   "Unit1.Em7.ControlNodes".sepaGripper."step".action1[330] := #_w1 AND NOT "Unit1.Em7.ControlNodes".cm.softCam.sepaGripperAxisX.avoidPos.inPos;
   "Unit1.Em7.ControlNodes".sepaGripper."step".transition1[330] := #_w1 AND "Unit1.Em7.ControlNodes".cm.softCam.sepaGripperAxisX.avoidPos.inPos;
   #statTonTime[330].TON(IN := #_w1 AND "Unit1.Em7.ControlNodes".sepaGripper."step".transition1[330],
                         PT := T#1000ms);
   IF #statTonTime[330].Q THEN
       "Unit1.Em7.ControlNodes".sepaGripper.sequence.status.nextStep := #JOB_3_STEP_90;
   END_IF;
END_REGION

REGION Network 32: Step[390] : Job[3] Step End
   RUNG wire#powerrail
      { S7_Templates := "SrcType := DInt" } EQ_Contact(in1 := "Unit1.Em7.ControlNodes".sepaGripper.sequence.status.currentStep, in2 := #JOB_3_STEP_90)
      Contact( "Unit1.Em7.ControlNodes".sepaGripper.sequence.status.seqActive )
      wire#w1
      Coil( "Unit1.Em7.ControlNodes".sepaGripper."step".action1[390] )
   END_RUNG
   RUNG wire#w1
      Coil( "Unit1.Em7.ControlNodes".sepaGripper."step".transition1[390] )
   END_RUNG
   RUNG wire#w1
      Contact( "Unit1.Em7.ControlNodes".sepaGripper."step".transition1[390] )
      { S7_Templates := "time_type := Time" } #statTonTime[390].TON(pt := T#1000ms, et =>)
      Move(in := #STEP_IDLE, out1 => "Unit1.Em7.ControlNodes".sepaGripper.sequence.status.nextStep)
   END_RUNG
   // the same network as SCL:
   "Unit1.Em7.ControlNodes".sepaGripper."step".action1[390] := ("Unit1.Em7.ControlNodes".sepaGripper.sequence.status.currentStep = #JOB_3_STEP_90) AND "Unit1.Em7.ControlNodes".sepaGripper.sequence.status.seqActive;
   "Unit1.Em7.ControlNodes".sepaGripper."step".transition1[390] := ("Unit1.Em7.ControlNodes".sepaGripper.sequence.status.currentStep = #JOB_3_STEP_90) AND "Unit1.Em7.ControlNodes".sepaGripper.sequence.status.seqActive;
   #statTonTime[390].TON(IN := ("Unit1.Em7.ControlNodes".sepaGripper.sequence.status.currentStep = #JOB_3_STEP_90) AND "Unit1.Em7.ControlNodes".sepaGripper.sequence.status.seqActive AND "Unit1.Em7.ControlNodes".sepaGripper."step".transition1[390],
                         PT := T#1000ms);
   IF #statTonTime[390].Q THEN
       "Unit1.Em7.ControlNodes".sepaGripper.sequence.status.nextStep := #STEP_IDLE;
   END_IF;
END_REGION

REGION Network 33: ******************** JOB[4] Reload ********************
END_REGION

REGION Network 34: Step[401] : JOB[4] Condition
   RUNG wire#powerrail
      { S7_Templates := "SrcType := DInt" } EQ_Contact(in1 := "Unit1.Em7.ControlNodes".sepaGripper.sequence.status.currentStep, in2 := #JOB_4_STEP_01)
      Contact( "Unit1.Em7.ControlNodes".sepaGripper.sequence.status.seqActive )
      wire#w1
      Coil( "Unit1.Em7.ControlNodes".sepaGripper."step".action1[401] )
   END_RUNG
   RUNG wire#w1
      Coil( "Unit1.Em7.ControlNodes".sepaGripper."step".transition1[401] )
   END_RUNG
   RUNG wire#w1
      Contact( "Unit1.Em7.ControlNodes".sepaGripper."step".transition1[401] )
      { S7_Templates := "time_type := Time" } #statTonTime[401].TON(pt := T#1000ms, et =>)
      Move(in := #JOB_4_STEP_10, out1 => "Unit1.Em7.ControlNodes".sepaGripper.sequence.status.nextStep)
   END_RUNG
   // the same network as SCL:
   "Unit1.Em7.ControlNodes".sepaGripper."step".action1[401] := ("Unit1.Em7.ControlNodes".sepaGripper.sequence.status.currentStep = #JOB_4_STEP_01) AND "Unit1.Em7.ControlNodes".sepaGripper.sequence.status.seqActive;
   "Unit1.Em7.ControlNodes".sepaGripper."step".transition1[401] := ("Unit1.Em7.ControlNodes".sepaGripper.sequence.status.currentStep = #JOB_4_STEP_01) AND "Unit1.Em7.ControlNodes".sepaGripper.sequence.status.seqActive;
   #statTonTime[401].TON(IN := ("Unit1.Em7.ControlNodes".sepaGripper.sequence.status.currentStep = #JOB_4_STEP_01) AND "Unit1.Em7.ControlNodes".sepaGripper.sequence.status.seqActive AND "Unit1.Em7.ControlNodes".sepaGripper."step".transition1[401],
                         PT := T#1000ms);
   IF #statTonTime[401].Q THEN
       "Unit1.Em7.ControlNodes".sepaGripper.sequence.status.nextStep := #JOB_4_STEP_10;
   END_IF;
END_REGION

REGION Network 35: Step[410] : Gripper X,Z-Axis Reload Pos
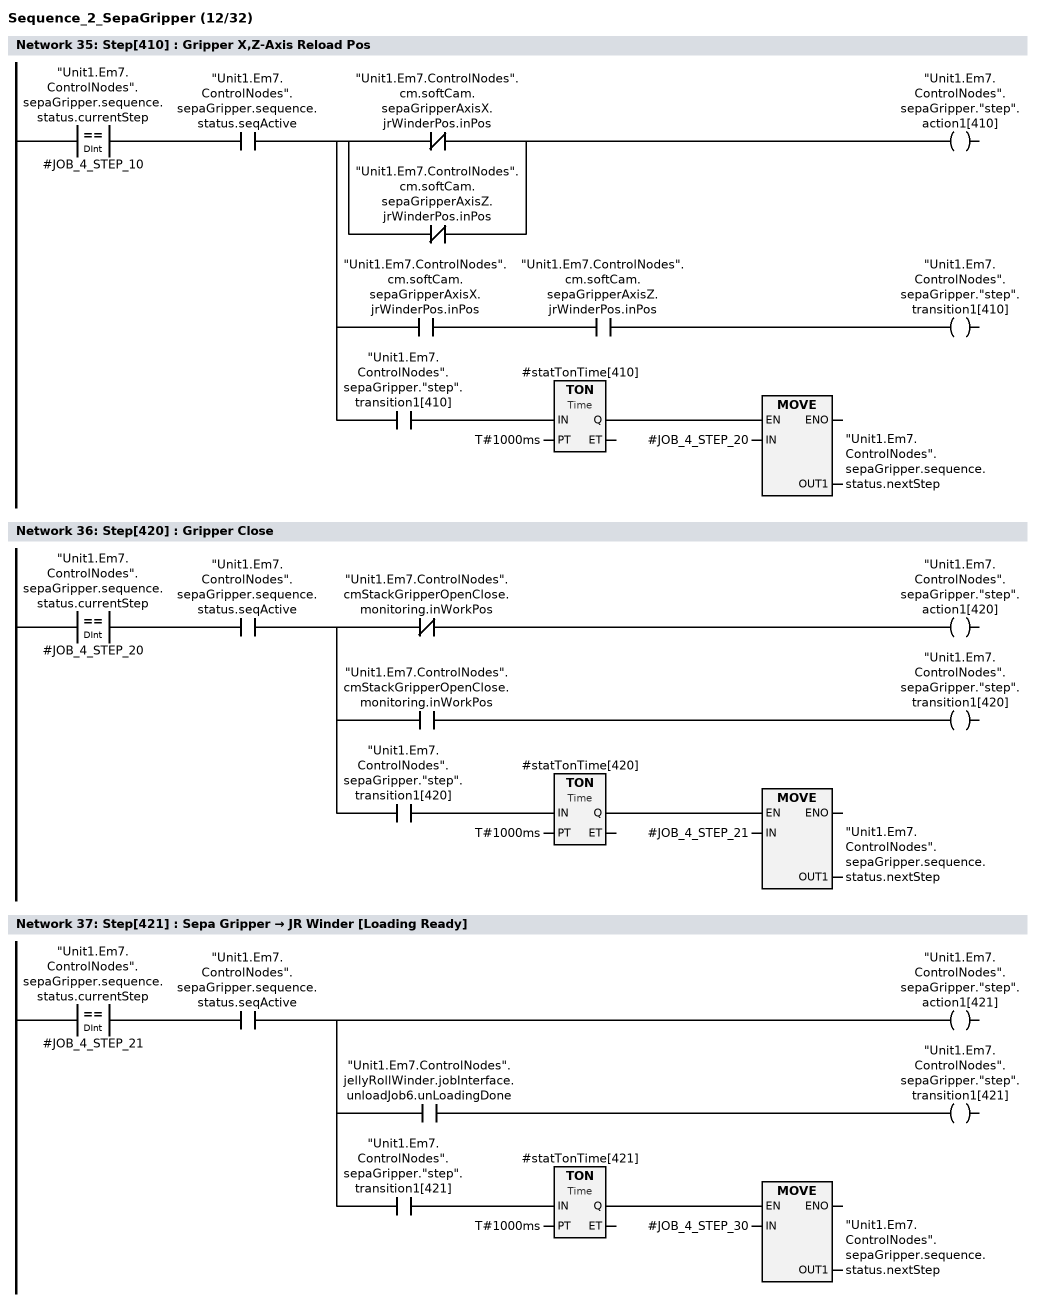
   RUNG wire#powerrail
      { S7_Templates := "SrcType := DInt" } EQ_Contact(in1 := "Unit1.Em7.ControlNodes".sepaGripper.sequence.status.currentStep, in2 := #JOB_4_STEP_10)
      Contact( "Unit1.Em7.ControlNodes".sepaGripper.sequence.status.seqActive )
      wire#w1
      I_Contact( "Unit1.Em7.ControlNodes".cm.softCam.sepaGripperAxisX.jrWinderPos.inPos )
      wire#w2
      Coil( "Unit1.Em7.ControlNodes".sepaGripper."step".action1[410] )
   END_RUNG
   RUNG wire#w1
      I_Contact( "Unit1.Em7.ControlNodes".cm.softCam.sepaGripperAxisZ.jrWinderPos.inPos )
   END_RUNG wire#w2
   RUNG wire#w1
      Contact( "Unit1.Em7.ControlNodes".cm.softCam.sepaGripperAxisX.jrWinderPos.inPos )
      Contact( "Unit1.Em7.ControlNodes".cm.softCam.sepaGripperAxisZ.jrWinderPos.inPos )
      Coil( "Unit1.Em7.ControlNodes".sepaGripper."step".transition1[410] )
   END_RUNG
   RUNG wire#w1
      Contact( "Unit1.Em7.ControlNodes".sepaGripper."step".transition1[410] )
      { S7_Templates := "time_type := Time" } #statTonTime[410].TON(pt := T#1000ms, et =>)
      Move(in := #JOB_4_STEP_20, out1 => "Unit1.Em7.ControlNodes".sepaGripper.sequence.status.nextStep)
   END_RUNG
   // the same network as SCL:
   #_w1 := ("Unit1.Em7.ControlNodes".sepaGripper.sequence.status.currentStep = #JOB_4_STEP_10) AND "Unit1.Em7.ControlNodes".sepaGripper.sequence.status.seqActive;
   "Unit1.Em7.ControlNodes".sepaGripper."step".action1[410] := #_w1 AND (NOT "Unit1.Em7.ControlNodes".cm.softCam.sepaGripperAxisX.jrWinderPos.inPos OR NOT "Unit1.Em7.ControlNodes".cm.softCam.sepaGripperAxisZ.jrWinderPos.inPos);
   "Unit1.Em7.ControlNodes".sepaGripper."step".transition1[410] := #_w1 AND "Unit1.Em7.ControlNodes".cm.softCam.sepaGripperAxisX.jrWinderPos.inPos AND "Unit1.Em7.ControlNodes".cm.softCam.sepaGripperAxisZ.jrWinderPos.inPos;
   #statTonTime[410].TON(IN := #_w1 AND "Unit1.Em7.ControlNodes".sepaGripper."step".transition1[410],
                         PT := T#1000ms);
   IF #statTonTime[410].Q THEN
       "Unit1.Em7.ControlNodes".sepaGripper.sequence.status.nextStep := #JOB_4_STEP_20;
   END_IF;
END_REGION

REGION Network 36: Step[420] : Gripper Close
   RUNG wire#powerrail
      { S7_Templates := "SrcType := DInt" } EQ_Contact(in1 := "Unit1.Em7.ControlNodes".sepaGripper.sequence.status.currentStep, in2 := #JOB_4_STEP_20)
      Contact( "Unit1.Em7.ControlNodes".sepaGripper.sequence.status.seqActive )
      wire#w1
      I_Contact( "Unit1.Em7.ControlNodes".cmStackGripperOpenClose.monitoring.inWorkPos )
      Coil( "Unit1.Em7.ControlNodes".sepaGripper."step".action1[420] )
   END_RUNG
   RUNG wire#w1
      Contact( "Unit1.Em7.ControlNodes".cmStackGripperOpenClose.monitoring.inWorkPos )
      Coil( "Unit1.Em7.ControlNodes".sepaGripper."step".transition1[420] )
   END_RUNG
   RUNG wire#w1
      Contact( "Unit1.Em7.ControlNodes".sepaGripper."step".transition1[420] )
      { S7_Templates := "time_type := Time" } #statTonTime[420].TON(pt := T#1000ms, et =>)
      Move(in := #JOB_4_STEP_21, out1 => "Unit1.Em7.ControlNodes".sepaGripper.sequence.status.nextStep)
   END_RUNG
   // the same network as SCL:
   #_w1 := ("Unit1.Em7.ControlNodes".sepaGripper.sequence.status.currentStep = #JOB_4_STEP_20) AND "Unit1.Em7.ControlNodes".sepaGripper.sequence.status.seqActive;
   "Unit1.Em7.ControlNodes".sepaGripper."step".action1[420] := #_w1 AND NOT "Unit1.Em7.ControlNodes".cmStackGripperOpenClose.monitoring.inWorkPos;
   "Unit1.Em7.ControlNodes".sepaGripper."step".transition1[420] := #_w1 AND "Unit1.Em7.ControlNodes".cmStackGripperOpenClose.monitoring.inWorkPos;
   #statTonTime[420].TON(IN := #_w1 AND "Unit1.Em7.ControlNodes".sepaGripper."step".transition1[420],
                         PT := T#1000ms);
   IF #statTonTime[420].Q THEN
       "Unit1.Em7.ControlNodes".sepaGripper.sequence.status.nextStep := #JOB_4_STEP_21;
   END_IF;
END_REGION

REGION Network 37: Step[421] : Sepa Gripper → JR Winder [Loading Ready]
   RUNG wire#powerrail
      { S7_Templates := "SrcType := DInt" } EQ_Contact(in1 := "Unit1.Em7.ControlNodes".sepaGripper.sequence.status.currentStep, in2 := #JOB_4_STEP_21)
      Contact( "Unit1.Em7.ControlNodes".sepaGripper.sequence.status.seqActive )
      wire#w1
      Coil( "Unit1.Em7.ControlNodes".sepaGripper."step".action1[421] )
   END_RUNG
   RUNG wire#w1
      Contact( "Unit1.Em7.ControlNodes".jellyRollWinder.jobInterface.unloadJob6.unLoadingDone )
      Coil( "Unit1.Em7.ControlNodes".sepaGripper."step".transition1[421] )
   END_RUNG
   RUNG wire#w1
      Contact( "Unit1.Em7.ControlNodes".sepaGripper."step".transition1[421] )
      { S7_Templates := "time_type := Time" } #statTonTime[421].TON(pt := T#1000ms, et =>)
      Move(in := #JOB_4_STEP_30, out1 => "Unit1.Em7.ControlNodes".sepaGripper.sequence.status.nextStep)
   END_RUNG
   // the same network as SCL:
   "Unit1.Em7.ControlNodes".sepaGripper."step".action1[421] := ("Unit1.Em7.ControlNodes".sepaGripper.sequence.status.currentStep = #JOB_4_STEP_21) AND "Unit1.Em7.ControlNodes".sepaGripper.sequence.status.seqActive;
   "Unit1.Em7.ControlNodes".sepaGripper."step".transition1[421] := ("Unit1.Em7.ControlNodes".sepaGripper.sequence.status.currentStep = #JOB_4_STEP_21) AND "Unit1.Em7.ControlNodes".sepaGripper.sequence.status.seqActive AND "Unit1.Em7.ControlNodes".jellyRollWinder.jobInterface.unloadJob6.unLoadingDone;
   #statTonTime[421].TON(IN := ("Unit1.Em7.ControlNodes".sepaGripper.sequence.status.currentStep = #JOB_4_STEP_21) AND "Unit1.Em7.ControlNodes".sepaGripper.sequence.status.seqActive AND "Unit1.Em7.ControlNodes".sepaGripper."step".transition1[421],
                         PT := T#1000ms);
   IF #statTonTime[421].Q THEN
       "Unit1.Em7.ControlNodes".sepaGripper.sequence.status.nextStep := #JOB_4_STEP_30;
   END_IF;
END_REGION

REGION Network 38: Step[430] : Gripper X,Z-Axis Turn Pos
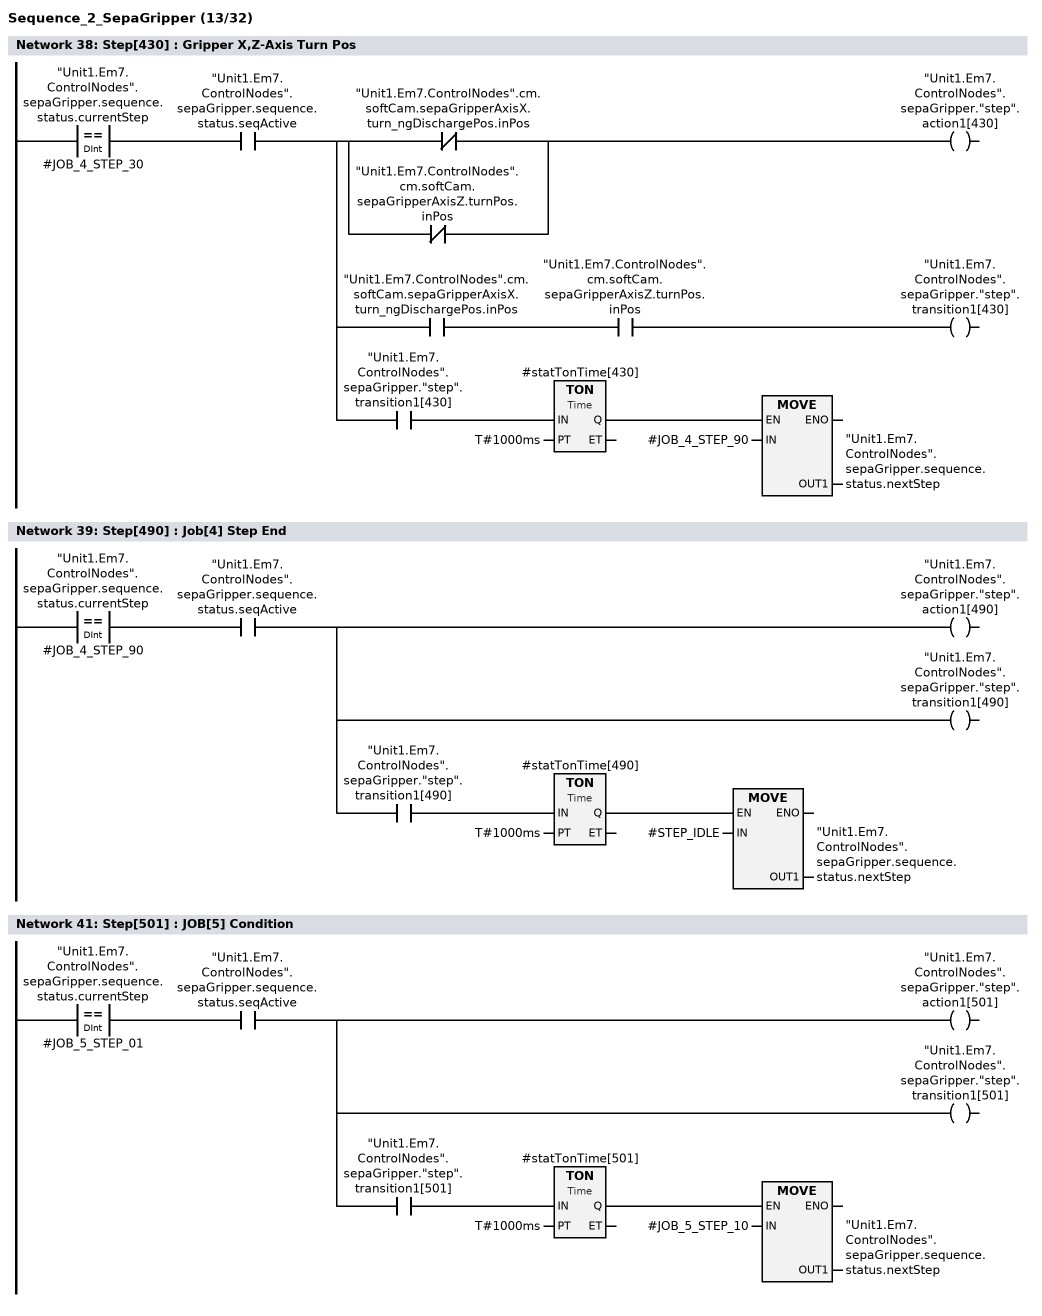
   RUNG wire#powerrail
      { S7_Templates := "SrcType := DInt" } EQ_Contact(in1 := "Unit1.Em7.ControlNodes".sepaGripper.sequence.status.currentStep, in2 := #JOB_4_STEP_30)
      Contact( "Unit1.Em7.ControlNodes".sepaGripper.sequence.status.seqActive )
      wire#w1
      I_Contact( "Unit1.Em7.ControlNodes".cm.softCam.sepaGripperAxisX.turn_ngDischargePos.inPos )
      wire#w2
      Coil( "Unit1.Em7.ControlNodes".sepaGripper."step".action1[430] )
   END_RUNG
   RUNG wire#w1
      I_Contact( "Unit1.Em7.ControlNodes".cm.softCam.sepaGripperAxisZ.turnPos.inPos )
   END_RUNG wire#w2
   RUNG wire#w1
      Contact( "Unit1.Em7.ControlNodes".cm.softCam.sepaGripperAxisX.turn_ngDischargePos.inPos )
      Contact( "Unit1.Em7.ControlNodes".cm.softCam.sepaGripperAxisZ.turnPos.inPos )
      Coil( "Unit1.Em7.ControlNodes".sepaGripper."step".transition1[430] )
   END_RUNG
   RUNG wire#w1
      Contact( "Unit1.Em7.ControlNodes".sepaGripper."step".transition1[430] )
      { S7_Templates := "time_type := Time" } #statTonTime[430].TON(pt := T#1000ms, et =>)
      Move(in := #JOB_4_STEP_90, out1 => "Unit1.Em7.ControlNodes".sepaGripper.sequence.status.nextStep)
   END_RUNG
   // the same network as SCL:
   #_w1 := ("Unit1.Em7.ControlNodes".sepaGripper.sequence.status.currentStep = #JOB_4_STEP_30) AND "Unit1.Em7.ControlNodes".sepaGripper.sequence.status.seqActive;
   "Unit1.Em7.ControlNodes".sepaGripper."step".action1[430] := #_w1 AND (NOT "Unit1.Em7.ControlNodes".cm.softCam.sepaGripperAxisX.turn_ngDischargePos.inPos OR NOT "Unit1.Em7.ControlNodes".cm.softCam.sepaGripperAxisZ.turnPos.inPos);
   "Unit1.Em7.ControlNodes".sepaGripper."step".transition1[430] := #_w1 AND "Unit1.Em7.ControlNodes".cm.softCam.sepaGripperAxisX.turn_ngDischargePos.inPos AND "Unit1.Em7.ControlNodes".cm.softCam.sepaGripperAxisZ.turnPos.inPos;
   #statTonTime[430].TON(IN := #_w1 AND "Unit1.Em7.ControlNodes".sepaGripper."step".transition1[430],
                         PT := T#1000ms);
   IF #statTonTime[430].Q THEN
       "Unit1.Em7.ControlNodes".sepaGripper.sequence.status.nextStep := #JOB_4_STEP_90;
   END_IF;
END_REGION

REGION Network 39: Step[490] : Job[4] Step End
   RUNG wire#powerrail
      { S7_Templates := "SrcType := DInt" } EQ_Contact(in1 := "Unit1.Em7.ControlNodes".sepaGripper.sequence.status.currentStep, in2 := #JOB_4_STEP_90)
      Contact( "Unit1.Em7.ControlNodes".sepaGripper.sequence.status.seqActive )
      wire#w1
      Coil( "Unit1.Em7.ControlNodes".sepaGripper."step".action1[490] )
   END_RUNG
   RUNG wire#w1
      Coil( "Unit1.Em7.ControlNodes".sepaGripper."step".transition1[490] )
   END_RUNG
   RUNG wire#w1
      Contact( "Unit1.Em7.ControlNodes".sepaGripper."step".transition1[490] )
      { S7_Templates := "time_type := Time" } #statTonTime[490].TON(pt := T#1000ms, et =>)
      Move(in := #STEP_IDLE, out1 => "Unit1.Em7.ControlNodes".sepaGripper.sequence.status.nextStep)
   END_RUNG
   // the same network as SCL:
   "Unit1.Em7.ControlNodes".sepaGripper."step".action1[490] := ("Unit1.Em7.ControlNodes".sepaGripper.sequence.status.currentStep = #JOB_4_STEP_90) AND "Unit1.Em7.ControlNodes".sepaGripper.sequence.status.seqActive;
   "Unit1.Em7.ControlNodes".sepaGripper."step".transition1[490] := ("Unit1.Em7.ControlNodes".sepaGripper.sequence.status.currentStep = #JOB_4_STEP_90) AND "Unit1.Em7.ControlNodes".sepaGripper.sequence.status.seqActive;
   #statTonTime[490].TON(IN := ("Unit1.Em7.ControlNodes".sepaGripper.sequence.status.currentStep = #JOB_4_STEP_90) AND "Unit1.Em7.ControlNodes".sepaGripper.sequence.status.seqActive AND "Unit1.Em7.ControlNodes".sepaGripper."step".transition1[490],
                         PT := T#1000ms);
   IF #statTonTime[490].Q THEN
       "Unit1.Em7.ControlNodes".sepaGripper.sequence.status.nextStep := #STEP_IDLE;
   END_IF;
END_REGION

REGION Network 40: ******************** JOB[5] UnReload ********************
END_REGION

REGION Network 41: Step[501] : JOB[5] Condition
   RUNG wire#powerrail
      { S7_Templates := "SrcType := DInt" } EQ_Contact(in1 := "Unit1.Em7.ControlNodes".sepaGripper.sequence.status.currentStep, in2 := #JOB_5_STEP_01)
      Contact( "Unit1.Em7.ControlNodes".sepaGripper.sequence.status.seqActive )
      wire#w1
      Coil( "Unit1.Em7.ControlNodes".sepaGripper."step".action1[501] )
   END_RUNG
   RUNG wire#w1
      Coil( "Unit1.Em7.ControlNodes".sepaGripper."step".transition1[501] )
   END_RUNG
   RUNG wire#w1
      Contact( "Unit1.Em7.ControlNodes".sepaGripper."step".transition1[501] )
      { S7_Templates := "time_type := Time" } #statTonTime[501].TON(pt := T#1000ms, et =>)
      Move(in := #JOB_5_STEP_10, out1 => "Unit1.Em7.ControlNodes".sepaGripper.sequence.status.nextStep)
   END_RUNG
   // the same network as SCL:
   "Unit1.Em7.ControlNodes".sepaGripper."step".action1[501] := ("Unit1.Em7.ControlNodes".sepaGripper.sequence.status.currentStep = #JOB_5_STEP_01) AND "Unit1.Em7.ControlNodes".sepaGripper.sequence.status.seqActive;
   "Unit1.Em7.ControlNodes".sepaGripper."step".transition1[501] := ("Unit1.Em7.ControlNodes".sepaGripper.sequence.status.currentStep = #JOB_5_STEP_01) AND "Unit1.Em7.ControlNodes".sepaGripper.sequence.status.seqActive;
   #statTonTime[501].TON(IN := ("Unit1.Em7.ControlNodes".sepaGripper.sequence.status.currentStep = #JOB_5_STEP_01) AND "Unit1.Em7.ControlNodes".sepaGripper.sequence.status.seqActive AND "Unit1.Em7.ControlNodes".sepaGripper."step".transition1[501],
                         PT := T#1000ms);
   IF #statTonTime[501].Q THEN
       "Unit1.Em7.ControlNodes".sepaGripper.sequence.status.nextStep := #JOB_5_STEP_10;
   END_IF;
END_REGION

REGION Network 42: Step[510] : Sepa Gripper → Inspection [Unloading Ready]
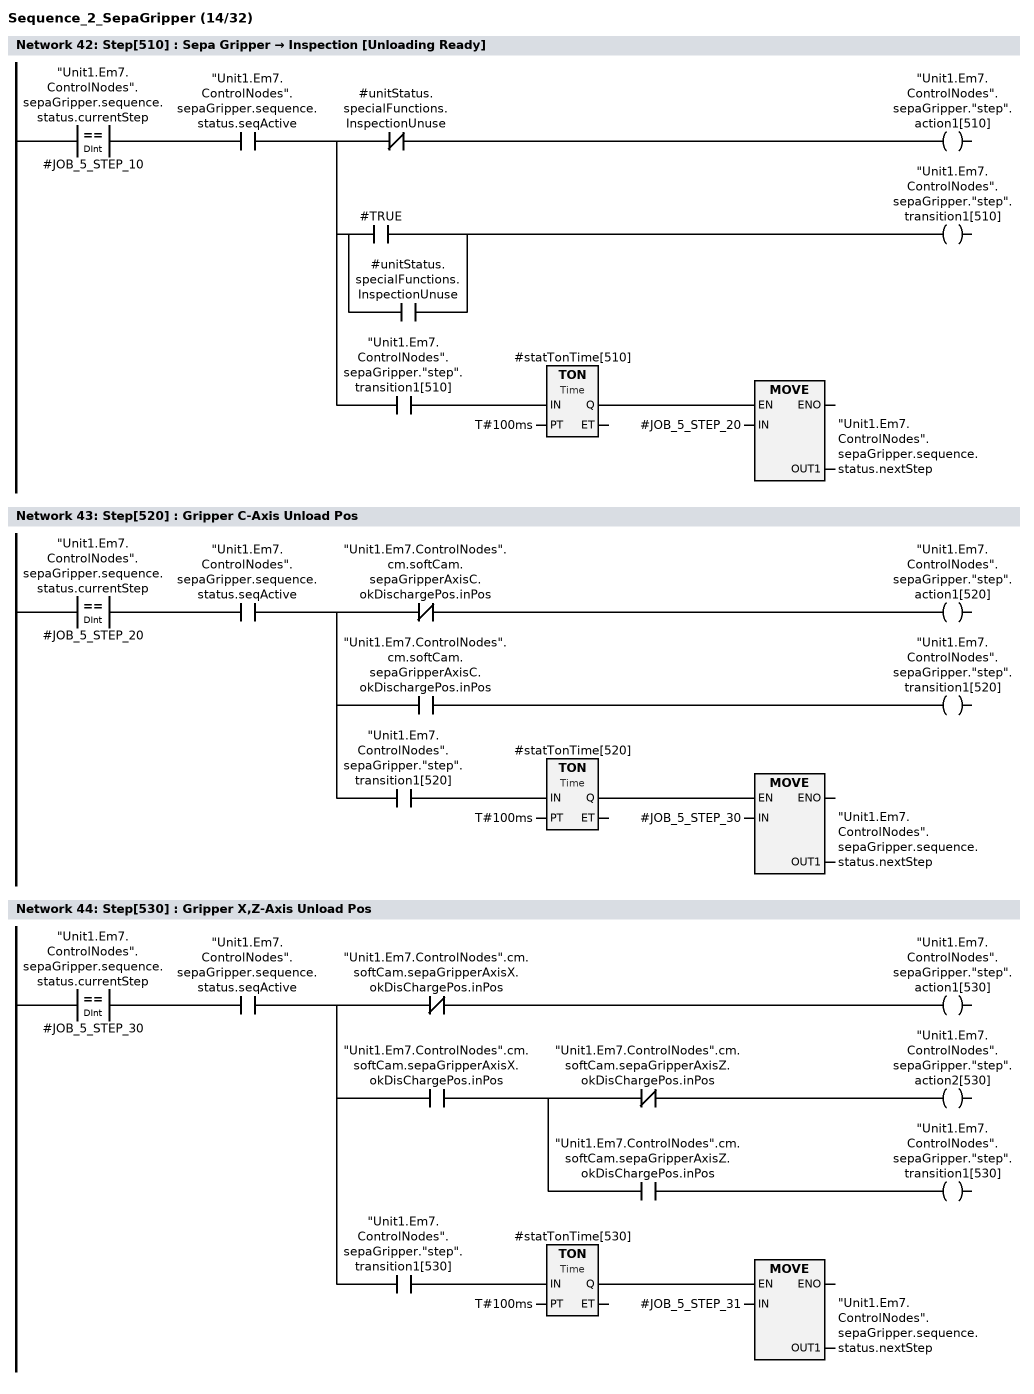
   RUNG wire#powerrail
      { S7_Templates := "SrcType := DInt" } EQ_Contact(in1 := "Unit1.Em7.ControlNodes".sepaGripper.sequence.status.currentStep, in2 := #JOB_5_STEP_10)
      Contact( "Unit1.Em7.ControlNodes".sepaGripper.sequence.status.seqActive )
      wire#w1
      I_Contact( #unitStatus.specialFunctions.InspectionUnuse )
      Coil( "Unit1.Em7.ControlNodes".sepaGripper."step".action1[510] )
   END_RUNG
   RUNG wire#w1
      Contact( #TRUE )
      wire#w2
      Coil( "Unit1.Em7.ControlNodes".sepaGripper."step".transition1[510] )
   END_RUNG
   RUNG wire#w1
      Contact( #unitStatus.specialFunctions.InspectionUnuse )
   END_RUNG wire#w2
   RUNG wire#w1
      Contact( "Unit1.Em7.ControlNodes".sepaGripper."step".transition1[510] )
      { S7_Templates := "time_type := Time" } #statTonTime[510].TON(pt := T#100ms, et =>)
      Move(in := #JOB_5_STEP_20, out1 => "Unit1.Em7.ControlNodes".sepaGripper.sequence.status.nextStep)
   END_RUNG
   // the same network as SCL:
   #_w1 := ("Unit1.Em7.ControlNodes".sepaGripper.sequence.status.currentStep = #JOB_5_STEP_10) AND "Unit1.Em7.ControlNodes".sepaGripper.sequence.status.seqActive;
   "Unit1.Em7.ControlNodes".sepaGripper."step".action1[510] := #_w1 AND NOT #unitStatus.specialFunctions.InspectionUnuse;
   "Unit1.Em7.ControlNodes".sepaGripper."step".transition1[510] := #_w1 AND (#TRUE OR #unitStatus.specialFunctions.InspectionUnuse);
   #statTonTime[510].TON(IN := #_w1 AND "Unit1.Em7.ControlNodes".sepaGripper."step".transition1[510],
                         PT := T#100ms);
   IF #statTonTime[510].Q THEN
       "Unit1.Em7.ControlNodes".sepaGripper.sequence.status.nextStep := #JOB_5_STEP_20;
   END_IF;
END_REGION

REGION Network 43: Step[520] : Gripper C-Axis Unload Pos
   RUNG wire#powerrail
      { S7_Templates := "SrcType := DInt" } EQ_Contact(in1 := "Unit1.Em7.ControlNodes".sepaGripper.sequence.status.currentStep, in2 := #JOB_5_STEP_20)
      Contact( "Unit1.Em7.ControlNodes".sepaGripper.sequence.status.seqActive )
      wire#w1
      I_Contact( "Unit1.Em7.ControlNodes".cm.softCam.sepaGripperAxisC.okDischargePos.inPos )
      Coil( "Unit1.Em7.ControlNodes".sepaGripper."step".action1[520] )
   END_RUNG
   RUNG wire#w1
      Contact( "Unit1.Em7.ControlNodes".cm.softCam.sepaGripperAxisC.okDischargePos.inPos )
      Coil( "Unit1.Em7.ControlNodes".sepaGripper."step".transition1[520] )
   END_RUNG
   RUNG wire#w1
      Contact( "Unit1.Em7.ControlNodes".sepaGripper."step".transition1[520] )
      { S7_Templates := "time_type := Time" } #statTonTime[520].TON(pt := T#100ms, et =>)
      Move(in := #JOB_5_STEP_30, out1 => "Unit1.Em7.ControlNodes".sepaGripper.sequence.status.nextStep)
   END_RUNG
   // the same network as SCL:
   #_w1 := ("Unit1.Em7.ControlNodes".sepaGripper.sequence.status.currentStep = #JOB_5_STEP_20) AND "Unit1.Em7.ControlNodes".sepaGripper.sequence.status.seqActive;
   "Unit1.Em7.ControlNodes".sepaGripper."step".action1[520] := #_w1 AND NOT "Unit1.Em7.ControlNodes".cm.softCam.sepaGripperAxisC.okDischargePos.inPos;
   "Unit1.Em7.ControlNodes".sepaGripper."step".transition1[520] := #_w1 AND "Unit1.Em7.ControlNodes".cm.softCam.sepaGripperAxisC.okDischargePos.inPos;
   #statTonTime[520].TON(IN := #_w1 AND "Unit1.Em7.ControlNodes".sepaGripper."step".transition1[520],
                         PT := T#100ms);
   IF #statTonTime[520].Q THEN
       "Unit1.Em7.ControlNodes".sepaGripper.sequence.status.nextStep := #JOB_5_STEP_30;
   END_IF;
END_REGION

REGION Network 44: Step[530] : Gripper X,Z-Axis Unload Pos
   RUNG wire#powerrail
      { S7_Templates := "SrcType := DInt" } EQ_Contact(in1 := "Unit1.Em7.ControlNodes".sepaGripper.sequence.status.currentStep, in2 := #JOB_5_STEP_30)
      Contact( "Unit1.Em7.ControlNodes".sepaGripper.sequence.status.seqActive )
      wire#w1
      I_Contact( "Unit1.Em7.ControlNodes".cm.softCam.sepaGripperAxisX.okDisChargePos.inPos )
      Coil( "Unit1.Em7.ControlNodes".sepaGripper."step".action1[530] )
   END_RUNG
   RUNG wire#w1
      Contact( "Unit1.Em7.ControlNodes".cm.softCam.sepaGripperAxisX.okDisChargePos.inPos )
      wire#w2
      I_Contact( "Unit1.Em7.ControlNodes".cm.softCam.sepaGripperAxisZ.okDisChargePos.inPos )
      Coil( "Unit1.Em7.ControlNodes".sepaGripper."step".action2[530] )
   END_RUNG
   RUNG wire#w2
      Contact( "Unit1.Em7.ControlNodes".cm.softCam.sepaGripperAxisZ.okDisChargePos.inPos )
      Coil( "Unit1.Em7.ControlNodes".sepaGripper."step".transition1[530] )
   END_RUNG
   RUNG wire#w1
      Contact( "Unit1.Em7.ControlNodes".sepaGripper."step".transition1[530] )
      { S7_Templates := "time_type := Time" } #statTonTime[530].TON(pt := T#100ms, et =>)
      Move(in := #JOB_5_STEP_31, out1 => "Unit1.Em7.ControlNodes".sepaGripper.sequence.status.nextStep)
   END_RUNG
   // the same network as SCL:
   #_w1 := ("Unit1.Em7.ControlNodes".sepaGripper.sequence.status.currentStep = #JOB_5_STEP_30) AND "Unit1.Em7.ControlNodes".sepaGripper.sequence.status.seqActive;
   "Unit1.Em7.ControlNodes".sepaGripper."step".action1[530] := #_w1 AND NOT "Unit1.Em7.ControlNodes".cm.softCam.sepaGripperAxisX.okDisChargePos.inPos;
   #_w2 := #_w1 AND "Unit1.Em7.ControlNodes".cm.softCam.sepaGripperAxisX.okDisChargePos.inPos;
   "Unit1.Em7.ControlNodes".sepaGripper."step".action2[530] := #_w2 AND NOT "Unit1.Em7.ControlNodes".cm.softCam.sepaGripperAxisZ.okDisChargePos.inPos;
   "Unit1.Em7.ControlNodes".sepaGripper."step".transition1[530] := #_w2 AND "Unit1.Em7.ControlNodes".cm.softCam.sepaGripperAxisZ.okDisChargePos.inPos;
   #statTonTime[530].TON(IN := #_w1 AND "Unit1.Em7.ControlNodes".sepaGripper."step".transition1[530],
                         PT := T#100ms);
   IF #statTonTime[530].Q THEN
       "Unit1.Em7.ControlNodes".sepaGripper.sequence.status.nextStep := #JOB_5_STEP_31;
   END_IF;
END_REGION

REGION Network 45: Step[531] : Sepa Gripper → Inspection [Clamp Request]
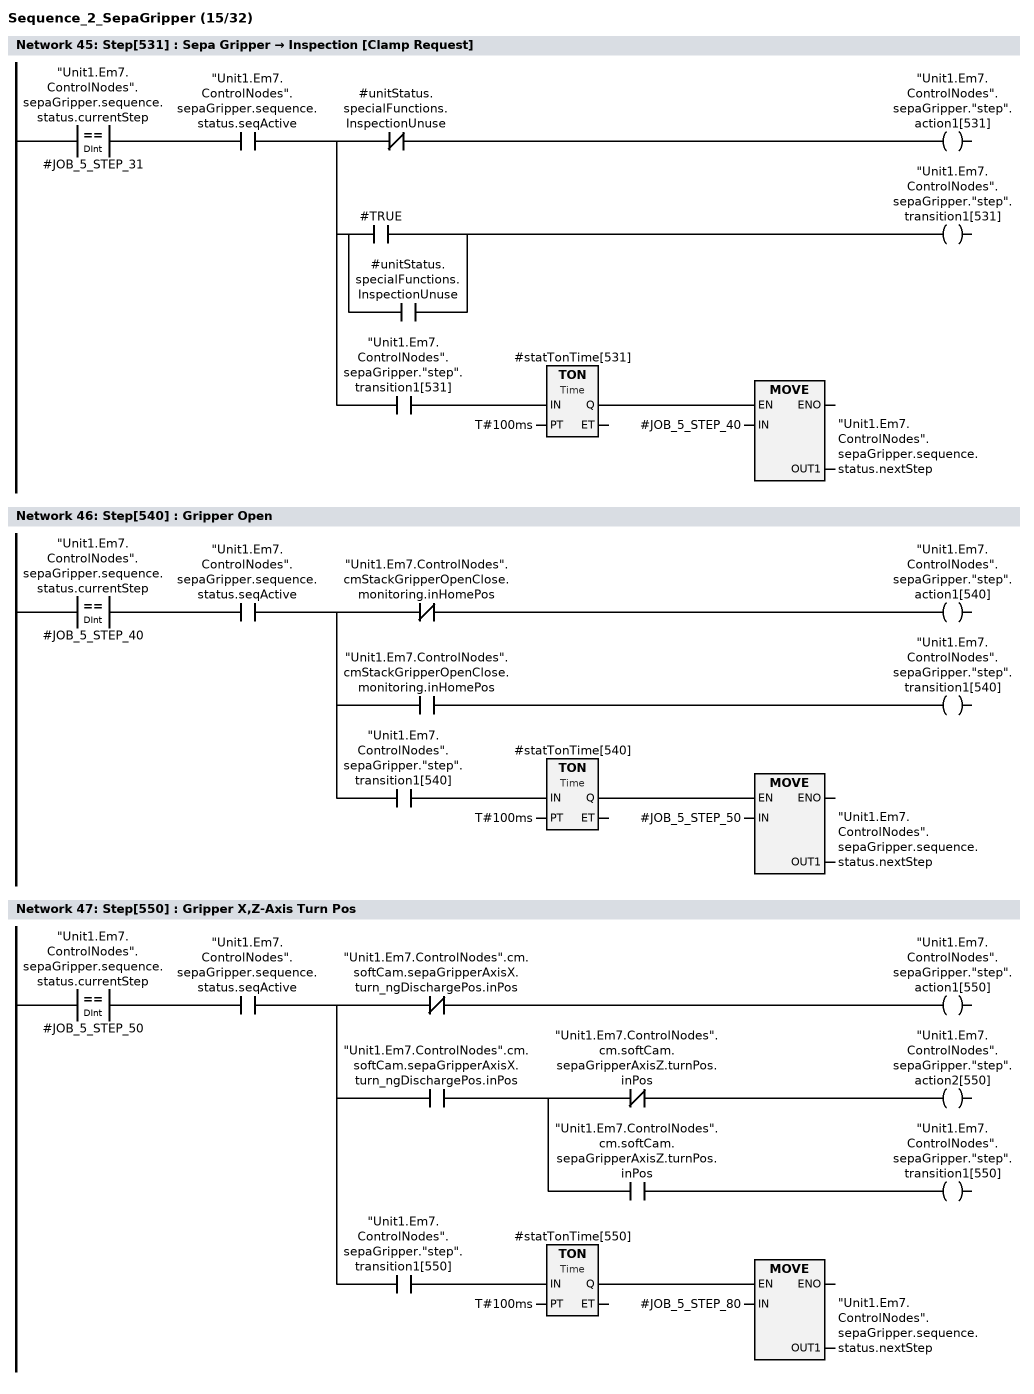
   RUNG wire#powerrail
      { S7_Templates := "SrcType := DInt" } EQ_Contact(in1 := "Unit1.Em7.ControlNodes".sepaGripper.sequence.status.currentStep, in2 := #JOB_5_STEP_31)
      Contact( "Unit1.Em7.ControlNodes".sepaGripper.sequence.status.seqActive )
      wire#w1
      I_Contact( #unitStatus.specialFunctions.InspectionUnuse )
      Coil( "Unit1.Em7.ControlNodes".sepaGripper."step".action1[531] )
   END_RUNG
   RUNG wire#w1
      Contact( #TRUE )
      wire#w2
      Coil( "Unit1.Em7.ControlNodes".sepaGripper."step".transition1[531] )
   END_RUNG
   RUNG wire#w1
      Contact( #unitStatus.specialFunctions.InspectionUnuse )
   END_RUNG wire#w2
   RUNG wire#w1
      Contact( "Unit1.Em7.ControlNodes".sepaGripper."step".transition1[531] )
      { S7_Templates := "time_type := Time" } #statTonTime[531].TON(pt := T#100ms, et =>)
      Move(in := #JOB_5_STEP_40, out1 => "Unit1.Em7.ControlNodes".sepaGripper.sequence.status.nextStep)
   END_RUNG
   // the same network as SCL:
   #_w1 := ("Unit1.Em7.ControlNodes".sepaGripper.sequence.status.currentStep = #JOB_5_STEP_31) AND "Unit1.Em7.ControlNodes".sepaGripper.sequence.status.seqActive;
   "Unit1.Em7.ControlNodes".sepaGripper."step".action1[531] := #_w1 AND NOT #unitStatus.specialFunctions.InspectionUnuse;
   "Unit1.Em7.ControlNodes".sepaGripper."step".transition1[531] := #_w1 AND (#TRUE OR #unitStatus.specialFunctions.InspectionUnuse);
   #statTonTime[531].TON(IN := #_w1 AND "Unit1.Em7.ControlNodes".sepaGripper."step".transition1[531],
                         PT := T#100ms);
   IF #statTonTime[531].Q THEN
       "Unit1.Em7.ControlNodes".sepaGripper.sequence.status.nextStep := #JOB_5_STEP_40;
   END_IF;
END_REGION

REGION Network 46: Step[540] : Gripper Open
   RUNG wire#powerrail
      { S7_Templates := "SrcType := DInt" } EQ_Contact(in1 := "Unit1.Em7.ControlNodes".sepaGripper.sequence.status.currentStep, in2 := #JOB_5_STEP_40)
      Contact( "Unit1.Em7.ControlNodes".sepaGripper.sequence.status.seqActive )
      wire#w1
      I_Contact( "Unit1.Em7.ControlNodes".cmStackGripperOpenClose.monitoring.inHomePos )
      Coil( "Unit1.Em7.ControlNodes".sepaGripper."step".action1[540] )
   END_RUNG
   RUNG wire#w1
      Contact( "Unit1.Em7.ControlNodes".cmStackGripperOpenClose.monitoring.inHomePos )
      Coil( "Unit1.Em7.ControlNodes".sepaGripper."step".transition1[540] )
   END_RUNG
   RUNG wire#w1
      Contact( "Unit1.Em7.ControlNodes".sepaGripper."step".transition1[540] )
      { S7_Templates := "time_type := Time" } #statTonTime[540].TON(pt := T#100ms, et =>)
      Move(in := #JOB_5_STEP_50, out1 => "Unit1.Em7.ControlNodes".sepaGripper.sequence.status.nextStep)
   END_RUNG
   // the same network as SCL:
   #_w1 := ("Unit1.Em7.ControlNodes".sepaGripper.sequence.status.currentStep = #JOB_5_STEP_40) AND "Unit1.Em7.ControlNodes".sepaGripper.sequence.status.seqActive;
   "Unit1.Em7.ControlNodes".sepaGripper."step".action1[540] := #_w1 AND NOT "Unit1.Em7.ControlNodes".cmStackGripperOpenClose.monitoring.inHomePos;
   "Unit1.Em7.ControlNodes".sepaGripper."step".transition1[540] := #_w1 AND "Unit1.Em7.ControlNodes".cmStackGripperOpenClose.monitoring.inHomePos;
   #statTonTime[540].TON(IN := #_w1 AND "Unit1.Em7.ControlNodes".sepaGripper."step".transition1[540],
                         PT := T#100ms);
   IF #statTonTime[540].Q THEN
       "Unit1.Em7.ControlNodes".sepaGripper.sequence.status.nextStep := #JOB_5_STEP_50;
   END_IF;
END_REGION

REGION Network 47: Step[550] : Gripper X,Z-Axis Turn Pos
   RUNG wire#powerrail
      { S7_Templates := "SrcType := DInt" } EQ_Contact(in1 := "Unit1.Em7.ControlNodes".sepaGripper.sequence.status.currentStep, in2 := #JOB_5_STEP_50)
      Contact( "Unit1.Em7.ControlNodes".sepaGripper.sequence.status.seqActive )
      wire#w1
      I_Contact( "Unit1.Em7.ControlNodes".cm.softCam.sepaGripperAxisX.turn_ngDischargePos.inPos )
      Coil( "Unit1.Em7.ControlNodes".sepaGripper."step".action1[550] )
   END_RUNG
   RUNG wire#w1
      Contact( "Unit1.Em7.ControlNodes".cm.softCam.sepaGripperAxisX.turn_ngDischargePos.inPos )
      wire#w2
      I_Contact( "Unit1.Em7.ControlNodes".cm.softCam.sepaGripperAxisZ.turnPos.inPos )
      Coil( "Unit1.Em7.ControlNodes".sepaGripper."step".action2[550] )
   END_RUNG
   RUNG wire#w2
      Contact( "Unit1.Em7.ControlNodes".cm.softCam.sepaGripperAxisZ.turnPos.inPos )
      Coil( "Unit1.Em7.ControlNodes".sepaGripper."step".transition1[550] )
   END_RUNG
   RUNG wire#w1
      Contact( "Unit1.Em7.ControlNodes".sepaGripper."step".transition1[550] )
      { S7_Templates := "time_type := Time" } #statTonTime[550].TON(pt := T#100ms, et =>)
      Move(in := #JOB_5_STEP_80, out1 => "Unit1.Em7.ControlNodes".sepaGripper.sequence.status.nextStep)
   END_RUNG
   // the same network as SCL:
   #_w1 := ("Unit1.Em7.ControlNodes".sepaGripper.sequence.status.currentStep = #JOB_5_STEP_50) AND "Unit1.Em7.ControlNodes".sepaGripper.sequence.status.seqActive;
   "Unit1.Em7.ControlNodes".sepaGripper."step".action1[550] := #_w1 AND NOT "Unit1.Em7.ControlNodes".cm.softCam.sepaGripperAxisX.turn_ngDischargePos.inPos;
   #_w2 := #_w1 AND "Unit1.Em7.ControlNodes".cm.softCam.sepaGripperAxisX.turn_ngDischargePos.inPos;
   "Unit1.Em7.ControlNodes".sepaGripper."step".action2[550] := #_w2 AND NOT "Unit1.Em7.ControlNodes".cm.softCam.sepaGripperAxisZ.turnPos.inPos;
   "Unit1.Em7.ControlNodes".sepaGripper."step".transition1[550] := #_w2 AND "Unit1.Em7.ControlNodes".cm.softCam.sepaGripperAxisZ.turnPos.inPos;
   #statTonTime[550].TON(IN := #_w1 AND "Unit1.Em7.ControlNodes".sepaGripper."step".transition1[550],
                         PT := T#100ms);
   IF #statTonTime[550].Q THEN
       "Unit1.Em7.ControlNodes".sepaGripper.sequence.status.nextStep := #JOB_5_STEP_80;
   END_IF;
END_REGION

REGION Network 48: Step[580] : Gripper X,Z,C-Axis Wait Pos
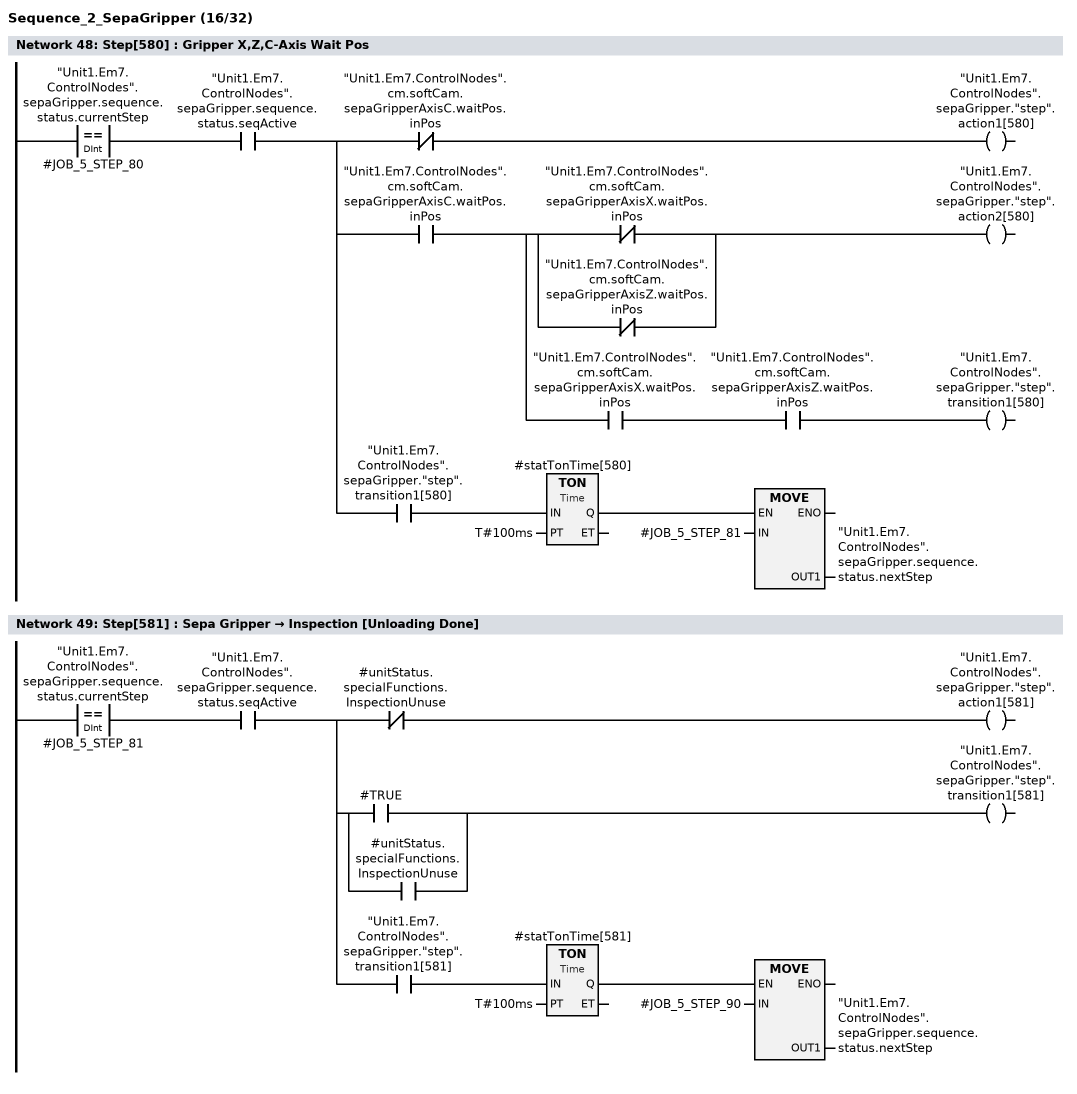
   RUNG wire#powerrail
      { S7_Templates := "SrcType := DInt" } EQ_Contact(in1 := "Unit1.Em7.ControlNodes".sepaGripper.sequence.status.currentStep, in2 := #JOB_5_STEP_80)
      Contact( "Unit1.Em7.ControlNodes".sepaGripper.sequence.status.seqActive )
      wire#w1
      I_Contact( "Unit1.Em7.ControlNodes".cm.softCam.sepaGripperAxisC.waitPos.inPos )
      Coil( "Unit1.Em7.ControlNodes".sepaGripper."step".action1[580] )
   END_RUNG
   RUNG wire#w1
      Contact( "Unit1.Em7.ControlNodes".cm.softCam.sepaGripperAxisC.waitPos.inPos )
      wire#w2
      I_Contact( "Unit1.Em7.ControlNodes".cm.softCam.sepaGripperAxisX.waitPos.inPos )
      wire#w3
      Coil( "Unit1.Em7.ControlNodes".sepaGripper."step".action2[580] )
   END_RUNG
   RUNG wire#w2
      I_Contact( "Unit1.Em7.ControlNodes".cm.softCam.sepaGripperAxisZ.waitPos.inPos )
   END_RUNG wire#w3
   RUNG wire#w2
      Contact( "Unit1.Em7.ControlNodes".cm.softCam.sepaGripperAxisX.waitPos.inPos )
      Contact( "Unit1.Em7.ControlNodes".cm.softCam.sepaGripperAxisZ.waitPos.inPos )
      Coil( "Unit1.Em7.ControlNodes".sepaGripper."step".transition1[580] )
   END_RUNG
   RUNG wire#w1
      Contact( "Unit1.Em7.ControlNodes".sepaGripper."step".transition1[580] )
      { S7_Templates := "time_type := Time" } #statTonTime[580].TON(pt := T#100ms, et =>)
      Move(in := #JOB_5_STEP_81, out1 => "Unit1.Em7.ControlNodes".sepaGripper.sequence.status.nextStep)
   END_RUNG
   // the same network as SCL:
   #_w1 := ("Unit1.Em7.ControlNodes".sepaGripper.sequence.status.currentStep = #JOB_5_STEP_80) AND "Unit1.Em7.ControlNodes".sepaGripper.sequence.status.seqActive;
   "Unit1.Em7.ControlNodes".sepaGripper."step".action1[580] := #_w1 AND NOT "Unit1.Em7.ControlNodes".cm.softCam.sepaGripperAxisC.waitPos.inPos;
   #_w2 := #_w1 AND "Unit1.Em7.ControlNodes".cm.softCam.sepaGripperAxisC.waitPos.inPos;
   "Unit1.Em7.ControlNodes".sepaGripper."step".action2[580] := #_w2 AND (NOT "Unit1.Em7.ControlNodes".cm.softCam.sepaGripperAxisX.waitPos.inPos OR NOT "Unit1.Em7.ControlNodes".cm.softCam.sepaGripperAxisZ.waitPos.inPos);
   "Unit1.Em7.ControlNodes".sepaGripper."step".transition1[580] := #_w2 AND "Unit1.Em7.ControlNodes".cm.softCam.sepaGripperAxisX.waitPos.inPos AND "Unit1.Em7.ControlNodes".cm.softCam.sepaGripperAxisZ.waitPos.inPos;
   #statTonTime[580].TON(IN := #_w1 AND "Unit1.Em7.ControlNodes".sepaGripper."step".transition1[580],
                         PT := T#100ms);
   IF #statTonTime[580].Q THEN
       "Unit1.Em7.ControlNodes".sepaGripper.sequence.status.nextStep := #JOB_5_STEP_81;
   END_IF;
END_REGION

REGION Network 49: Step[581] : Sepa Gripper → Inspection [Unloading Done]
   RUNG wire#powerrail
      { S7_Templates := "SrcType := DInt" } EQ_Contact(in1 := "Unit1.Em7.ControlNodes".sepaGripper.sequence.status.currentStep, in2 := #JOB_5_STEP_81)
      Contact( "Unit1.Em7.ControlNodes".sepaGripper.sequence.status.seqActive )
      wire#w1
      I_Contact( #unitStatus.specialFunctions.InspectionUnuse )
      Coil( "Unit1.Em7.ControlNodes".sepaGripper."step".action1[581] )
   END_RUNG
   RUNG wire#w1
      Contact( #TRUE )
      wire#w2
      Coil( "Unit1.Em7.ControlNodes".sepaGripper."step".transition1[581] )
   END_RUNG
   RUNG wire#w1
      Contact( #unitStatus.specialFunctions.InspectionUnuse )
   END_RUNG wire#w2
   RUNG wire#w1
      Contact( "Unit1.Em7.ControlNodes".sepaGripper."step".transition1[581] )
      { S7_Templates := "time_type := Time" } #statTonTime[581].TON(pt := T#100ms, et =>)
      Move(in := #JOB_5_STEP_90, out1 => "Unit1.Em7.ControlNodes".sepaGripper.sequence.status.nextStep)
   END_RUNG
   // the same network as SCL:
   #_w1 := ("Unit1.Em7.ControlNodes".sepaGripper.sequence.status.currentStep = #JOB_5_STEP_81) AND "Unit1.Em7.ControlNodes".sepaGripper.sequence.status.seqActive;
   "Unit1.Em7.ControlNodes".sepaGripper."step".action1[581] := #_w1 AND NOT #unitStatus.specialFunctions.InspectionUnuse;
   "Unit1.Em7.ControlNodes".sepaGripper."step".transition1[581] := #_w1 AND (#TRUE OR #unitStatus.specialFunctions.InspectionUnuse);
   #statTonTime[581].TON(IN := #_w1 AND "Unit1.Em7.ControlNodes".sepaGripper."step".transition1[581],
                         PT := T#100ms);
   IF #statTonTime[581].Q THEN
       "Unit1.Em7.ControlNodes".sepaGripper.sequence.status.nextStep := #JOB_5_STEP_90;
   END_IF;
END_REGION

REGION Network 50: Step[590] : Job[5] Step End
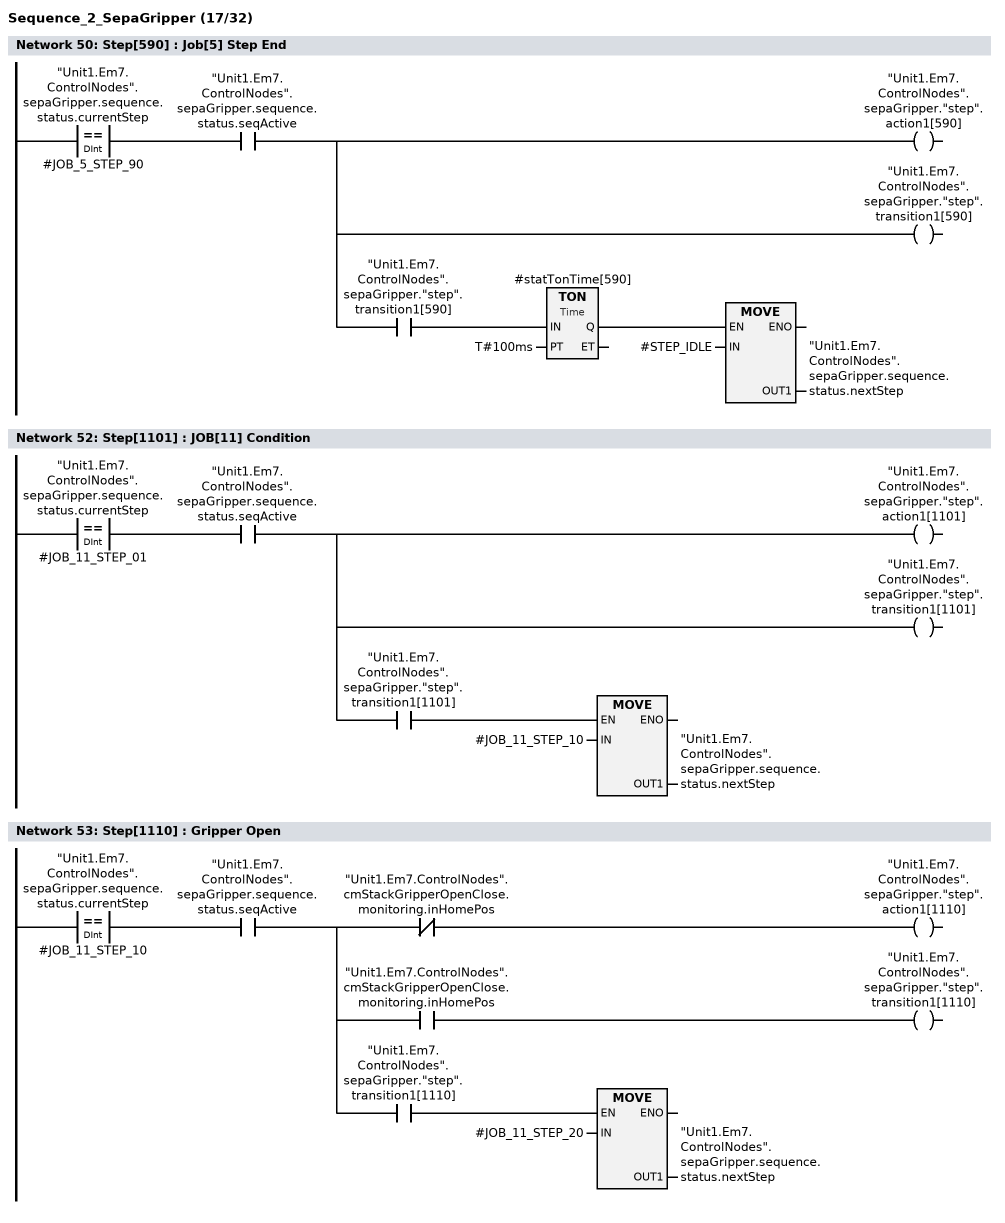
   RUNG wire#powerrail
      { S7_Templates := "SrcType := DInt" } EQ_Contact(in1 := "Unit1.Em7.ControlNodes".sepaGripper.sequence.status.currentStep, in2 := #JOB_5_STEP_90)
      Contact( "Unit1.Em7.ControlNodes".sepaGripper.sequence.status.seqActive )
      wire#w1
      Coil( "Unit1.Em7.ControlNodes".sepaGripper."step".action1[590] )
   END_RUNG
   RUNG wire#w1
      Coil( "Unit1.Em7.ControlNodes".sepaGripper."step".transition1[590] )
   END_RUNG
   RUNG wire#w1
      Contact( "Unit1.Em7.ControlNodes".sepaGripper."step".transition1[590] )
      { S7_Templates := "time_type := Time" } #statTonTime[590].TON(pt := T#100ms, et =>)
      Move(in := #STEP_IDLE, out1 => "Unit1.Em7.ControlNodes".sepaGripper.sequence.status.nextStep)
   END_RUNG
   // the same network as SCL:
   "Unit1.Em7.ControlNodes".sepaGripper."step".action1[590] := ("Unit1.Em7.ControlNodes".sepaGripper.sequence.status.currentStep = #JOB_5_STEP_90) AND "Unit1.Em7.ControlNodes".sepaGripper.sequence.status.seqActive;
   "Unit1.Em7.ControlNodes".sepaGripper."step".transition1[590] := ("Unit1.Em7.ControlNodes".sepaGripper.sequence.status.currentStep = #JOB_5_STEP_90) AND "Unit1.Em7.ControlNodes".sepaGripper.sequence.status.seqActive;
   #statTonTime[590].TON(IN := ("Unit1.Em7.ControlNodes".sepaGripper.sequence.status.currentStep = #JOB_5_STEP_90) AND "Unit1.Em7.ControlNodes".sepaGripper.sequence.status.seqActive AND "Unit1.Em7.ControlNodes".sepaGripper."step".transition1[590],
                         PT := T#100ms);
   IF #statTonTime[590].Q THEN
       "Unit1.Em7.ControlNodes".sepaGripper.sequence.status.nextStep := #STEP_IDLE;
   END_IF;
END_REGION

REGION Network 51: *************** IMMEDIATE STOP **************************
END_REGION

REGION Network 52: Step[1101] : JOB[11] Condition
   RUNG wire#powerrail
      { S7_Templates := "SrcType := DInt" } EQ_Contact(in1 := "Unit1.Em7.ControlNodes".sepaGripper.sequence.status.currentStep, in2 := #JOB_11_STEP_01)
      Contact( "Unit1.Em7.ControlNodes".sepaGripper.sequence.status.seqActive )
      wire#w1
      Coil( "Unit1.Em7.ControlNodes".sepaGripper."step".action1[1101] )
   END_RUNG
   RUNG wire#w1
      Coil( "Unit1.Em7.ControlNodes".sepaGripper."step".transition1[1101] )
   END_RUNG
   RUNG wire#w1
      Contact( "Unit1.Em7.ControlNodes".sepaGripper."step".transition1[1101] )
      Move(in := #JOB_11_STEP_10, out1 => "Unit1.Em7.ControlNodes".sepaGripper.sequence.status.nextStep)
   END_RUNG
   // the same network as SCL:
   "Unit1.Em7.ControlNodes".sepaGripper."step".action1[1101] := ("Unit1.Em7.ControlNodes".sepaGripper.sequence.status.currentStep = #JOB_11_STEP_01) AND "Unit1.Em7.ControlNodes".sepaGripper.sequence.status.seqActive;
   "Unit1.Em7.ControlNodes".sepaGripper."step".transition1[1101] := ("Unit1.Em7.ControlNodes".sepaGripper.sequence.status.currentStep = #JOB_11_STEP_01) AND "Unit1.Em7.ControlNodes".sepaGripper.sequence.status.seqActive;
   IF ("Unit1.Em7.ControlNodes".sepaGripper.sequence.status.currentStep = #JOB_11_STEP_01) AND "Unit1.Em7.ControlNodes".sepaGripper.sequence.status.seqActive AND "Unit1.Em7.ControlNodes".sepaGripper."step".transition1[1101] THEN
       "Unit1.Em7.ControlNodes".sepaGripper.sequence.status.nextStep := #JOB_11_STEP_10;
   END_IF;
END_REGION

REGION Network 53: Step[1110] : Gripper Open
   RUNG wire#powerrail
      { S7_Templates := "SrcType := DInt" } EQ_Contact(in1 := "Unit1.Em7.ControlNodes".sepaGripper.sequence.status.currentStep, in2 := #JOB_11_STEP_10)
      Contact( "Unit1.Em7.ControlNodes".sepaGripper.sequence.status.seqActive )
      wire#w1
      I_Contact( "Unit1.Em7.ControlNodes".cmStackGripperOpenClose.monitoring.inHomePos )
      Coil( "Unit1.Em7.ControlNodes".sepaGripper."step".action1[1110] )
   END_RUNG
   RUNG wire#w1
      Contact( "Unit1.Em7.ControlNodes".cmStackGripperOpenClose.monitoring.inHomePos )
      Coil( "Unit1.Em7.ControlNodes".sepaGripper."step".transition1[1110] )
   END_RUNG
   RUNG wire#w1
      Contact( "Unit1.Em7.ControlNodes".sepaGripper."step".transition1[1110] )
      Move(in := #JOB_11_STEP_20, out1 => "Unit1.Em7.ControlNodes".sepaGripper.sequence.status.nextStep)
   END_RUNG
   // the same network as SCL:
   #_w1 := ("Unit1.Em7.ControlNodes".sepaGripper.sequence.status.currentStep = #JOB_11_STEP_10) AND "Unit1.Em7.ControlNodes".sepaGripper.sequence.status.seqActive;
   "Unit1.Em7.ControlNodes".sepaGripper."step".action1[1110] := #_w1 AND NOT "Unit1.Em7.ControlNodes".cmStackGripperOpenClose.monitoring.inHomePos;
   "Unit1.Em7.ControlNodes".sepaGripper."step".transition1[1110] := #_w1 AND "Unit1.Em7.ControlNodes".cmStackGripperOpenClose.monitoring.inHomePos;
   IF #_w1 AND "Unit1.Em7.ControlNodes".sepaGripper."step".transition1[1110] THEN
       "Unit1.Em7.ControlNodes".sepaGripper.sequence.status.nextStep := #JOB_11_STEP_20;
   END_IF;
END_REGION

REGION Network 54: Step[1120] : Gripper X-Axis PickUp BeforePos
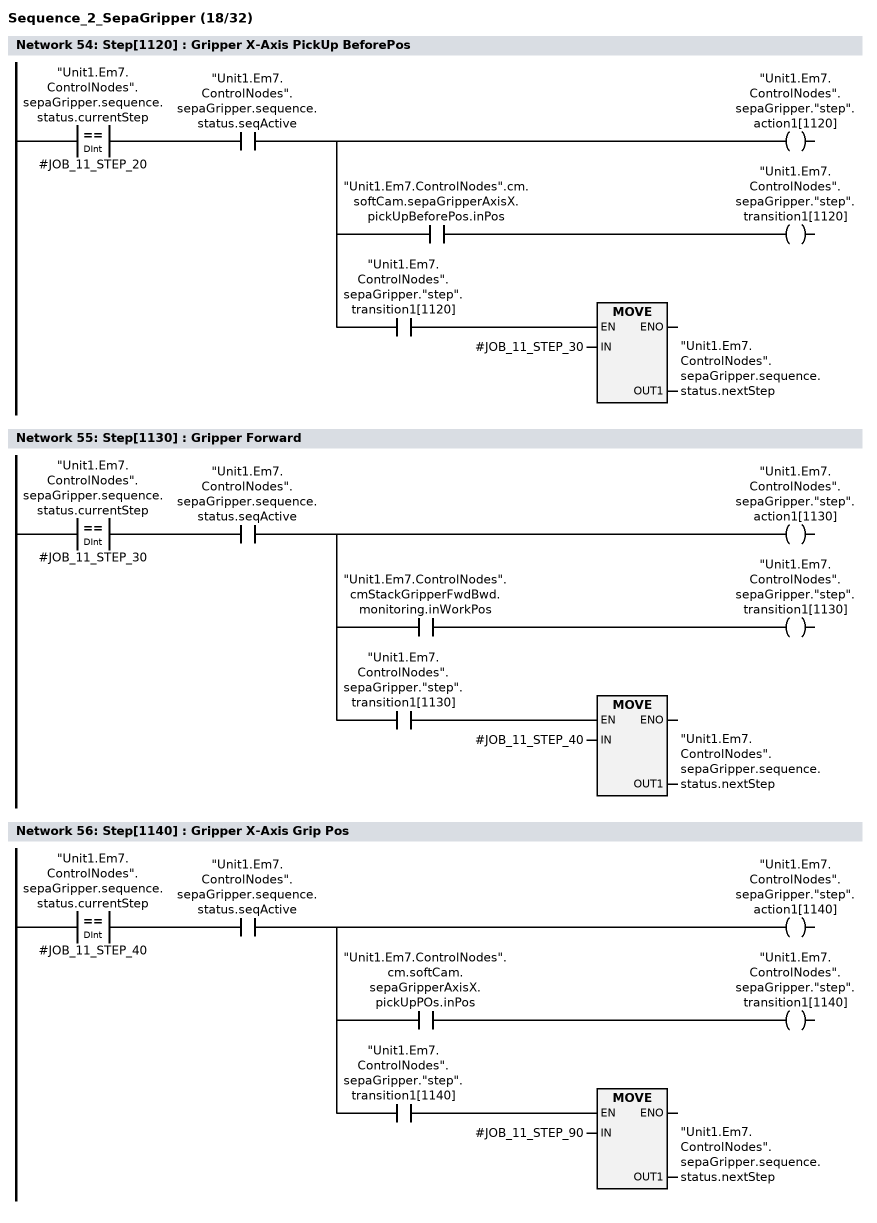
   RUNG wire#powerrail
      { S7_Templates := "SrcType := DInt" } EQ_Contact(in1 := "Unit1.Em7.ControlNodes".sepaGripper.sequence.status.currentStep, in2 := #JOB_11_STEP_20)
      Contact( "Unit1.Em7.ControlNodes".sepaGripper.sequence.status.seqActive )
      wire#w1
      Coil( "Unit1.Em7.ControlNodes".sepaGripper."step".action1[1120] )
   END_RUNG
   RUNG wire#w1
      Contact( "Unit1.Em7.ControlNodes".cm.softCam.sepaGripperAxisX.pickUpBeforePos.inPos )
      Coil( "Unit1.Em7.ControlNodes".sepaGripper."step".transition1[1120] )
   END_RUNG
   RUNG wire#w1
      Contact( "Unit1.Em7.ControlNodes".sepaGripper."step".transition1[1120] )
      Move(in := #JOB_11_STEP_30, out1 => "Unit1.Em7.ControlNodes".sepaGripper.sequence.status.nextStep)
   END_RUNG
   // the same network as SCL:
   "Unit1.Em7.ControlNodes".sepaGripper."step".action1[1120] := ("Unit1.Em7.ControlNodes".sepaGripper.sequence.status.currentStep = #JOB_11_STEP_20) AND "Unit1.Em7.ControlNodes".sepaGripper.sequence.status.seqActive;
   "Unit1.Em7.ControlNodes".sepaGripper."step".transition1[1120] := ("Unit1.Em7.ControlNodes".sepaGripper.sequence.status.currentStep = #JOB_11_STEP_20) AND "Unit1.Em7.ControlNodes".sepaGripper.sequence.status.seqActive AND "Unit1.Em7.ControlNodes".cm.softCam.sepaGripperAxisX.pickUpBeforePos.inPos;
   IF ("Unit1.Em7.ControlNodes".sepaGripper.sequence.status.currentStep = #JOB_11_STEP_20) AND "Unit1.Em7.ControlNodes".sepaGripper.sequence.status.seqActive AND "Unit1.Em7.ControlNodes".sepaGripper."step".transition1[1120] THEN
       "Unit1.Em7.ControlNodes".sepaGripper.sequence.status.nextStep := #JOB_11_STEP_30;
   END_IF;
END_REGION

REGION Network 55: Step[1130] : Gripper Forward
   RUNG wire#powerrail
      { S7_Templates := "SrcType := DInt" } EQ_Contact(in1 := "Unit1.Em7.ControlNodes".sepaGripper.sequence.status.currentStep, in2 := #JOB_11_STEP_30)
      Contact( "Unit1.Em7.ControlNodes".sepaGripper.sequence.status.seqActive )
      wire#w1
      Coil( "Unit1.Em7.ControlNodes".sepaGripper."step".action1[1130] )
   END_RUNG
   RUNG wire#w1
      Contact( "Unit1.Em7.ControlNodes".cmStackGripperFwdBwd.monitoring.inWorkPos )
      Coil( "Unit1.Em7.ControlNodes".sepaGripper."step".transition1[1130] )
   END_RUNG
   RUNG wire#w1
      Contact( "Unit1.Em7.ControlNodes".sepaGripper."step".transition1[1130] )
      Move(in := #JOB_11_STEP_40, out1 => "Unit1.Em7.ControlNodes".sepaGripper.sequence.status.nextStep)
   END_RUNG
   // the same network as SCL:
   "Unit1.Em7.ControlNodes".sepaGripper."step".action1[1130] := ("Unit1.Em7.ControlNodes".sepaGripper.sequence.status.currentStep = #JOB_11_STEP_30) AND "Unit1.Em7.ControlNodes".sepaGripper.sequence.status.seqActive;
   "Unit1.Em7.ControlNodes".sepaGripper."step".transition1[1130] := ("Unit1.Em7.ControlNodes".sepaGripper.sequence.status.currentStep = #JOB_11_STEP_30) AND "Unit1.Em7.ControlNodes".sepaGripper.sequence.status.seqActive AND "Unit1.Em7.ControlNodes".cmStackGripperFwdBwd.monitoring.inWorkPos;
   IF ("Unit1.Em7.ControlNodes".sepaGripper.sequence.status.currentStep = #JOB_11_STEP_30) AND "Unit1.Em7.ControlNodes".sepaGripper.sequence.status.seqActive AND "Unit1.Em7.ControlNodes".sepaGripper."step".transition1[1130] THEN
       "Unit1.Em7.ControlNodes".sepaGripper.sequence.status.nextStep := #JOB_11_STEP_40;
   END_IF;
END_REGION

